		IF NOT WriteAdsPara.BUSY
			AND NOT WriteAdsPara.WRITE
		 	AND NOT Error
		THEN
			IF (forceSoftLimit XOR status.0) OR NOT InitDone.0 THEN
				InitDone.0 									:= TRUE;
				status.0 									:= forceSoftLimit;
				tmpWord 									:= BOOL_TO_UINT(forceSoftLimit);
				State 										:= 1;
				Busy 										:= TRUE;

			ELSIF(forceCalibration XOR status.1) OR NOT InitDone.1 THEN
				InitDone.1 									:= TRUE;
				status.1 									:= forceCalibration;
				tmpWord 									:= BOOL_TO_UINT(forceCalibration);
				State 										:= 10;
				Busy 										:= TRUE;
	
			ELSIF(forcePosLagMon XOR status.2) OR NOT InitDone.2 THEN
				InitDone.2 									:= TRUE;
				status.2 									:= forcePosLagMon;
				tmpWord 									:= BOOL_TO_UINT(forcePosLagMon);
				State 										:= 20;
				Busy 										:= TRUE;
			ELSIF(forcePosMon XOR status.3) OR NOT InitDone.3 THEN
				InitDone.3 									:= TRUE;
				status.3 									:= forcePosMon;
				tmpWord 									:= BOOL_TO_UINT(forcePosMon);
				State 										:= 30;
				Busy 										:= TRUE;
			ELSIF(forceTargetMon XOR status.4) OR NOT InitDone.4 THEN
				InitDone.4 									:= TRUE;
				status.4 									:= forceTargetMon;
				tmpWord 									:= BOOL_TO_UINT(forceTargetMon);
				State 										:= 40;
				Busy 										:= TRUE;
		
			END_IF
		ELSE
			WriteAdsPara	(Write := FALSE);
		END_IF

	1: (* toggle positive limit switches ****************************************************************)
		IF NOT WriteAdsPara.Busy
			AND WriteAdsPara.Write
		THEN
			IF WriteAdsPara.Err THEN
				State 										:= 9999;  // goto Error-state 
			ELSE           									
				State 										:= State + 1;
			END_IF         	
		END_IF

		WriteAdsPara(
			IdxGrp	:=16#4000+AxisId,
			IdxOffs	:=16#1000C,
			LEN		:=SIZEOF(tmpWord),
			SrcAddr	:=ADR(tmpWord),
			Write 	:= State = 1);

	2: (* toggle negative limit switches *****************************************************************)
		IF NOT WriteAdsPara.Busy
			AND WriteAdsPara.Write
		THEN
			IF WriteAdsPara.Err THEN
				State 										:= 9999; // goto Error-state 
			ELSE
				State 										:= 99; // done 
			END_IF
		END_IF

		WriteAdsPara(
			IdxGrp	:=16#4000+AxisId,
			IdxOffs	:=16#1000B,
			LEN		:=SIZEOF(tmpWord),
			SrcAddr	:=ADR(tmpWord),
			Write 	:= State = 2);

	10: (* set referenceflag *****************************************************************)
		IF NOT WriteAdsPara.Busy
			AND WriteAdsPara.Write
		THEN
			IF WriteAdsPara.Err THEN
				State 										:= 9999;  	// goto Error-state 
			ELSE           									
				State 										:= 99; 		// done 
			END_IF
		END_IF

		WriteAdsPara(
			IdxGrp	:=16#5100+AxisId,
			IdxOffs	:=16#9,
			LEN		:=SIZEOF(tmpWord),
			SrcAddr	:=ADR(tmpWord),
			Write 	:= State = 10 );
			
	20: (* lagdistance monitoring *****************************************************************)
		IF NOT WriteAdsPara.Busy
			AND WriteAdsPara.Write
		THEN
			IF WriteAdsPara.Err THEN
				State 										:= 9999;  	// goto Error-state 
			ELSE           									
				State 										:= 99; 		// done
			END_IF
		END_IF

		WriteAdsPara(
			IdxGrp	:=16#6000+AxisId,
			IdxOffs	:=16#10,
			LEN		:=SIZEOF(tmpWord),
			SrcAddr	:=ADR(tmpWord),
			Write 	:= State = 20);
			
	30: (* Position Monitoring *****************************************************************)
		IF NOT WriteAdsPara.Busy
			AND WriteAdsPara.Write
		THEN
			IF WriteAdsPara.Err THEN
				State 										:= 9999;  	// goto Error-state 
			ELSE           									
				State 										:= 99; 		// done
			END_IF
		END_IF

		WriteAdsPara(

			IdxGrp	:=16#4000+AxisId,
			IdxOffs	:=16#F,
			LEN		:=SIZEOF(tmpWord),
			SrcAddr	:=ADR(tmpWord),
			Write 	:= State = 30 );

	40: (* Target Monitoring *****************************************************************)
		IF NOT WriteAdsPara.Busy
			AND WriteAdsPara.Write
		THEN
			IF WriteAdsPara.Err THEN
				State 										:= 9999;  	// goto Error-state 
			ELSE           									
				State 										:= 99; 		// done
			END_IF
		END_IF

		WriteAdsPara(
			IdxGrp	:=16#4000+AxisId,
			IdxOffs	:=16#15,
			LEN		:=SIZEOF(tmpWord),
			SrcAddr	:=ADR(tmpWord),
			Write 	:= State = 40 );
			
	ELSE (* case else *)
		IF WriteAdsPara.ERR THEN
			Error											:= TRUE;
			ErrorID											:= WriteAdsPara.ERRID;
			LastErrText										:= CONCAT('Err WriteAdsPara ID: ', UDINT_TO_STRING(ErrorID));
		ELSE            									
			State 											:= 0;
		END_IF
	END_CASE
END_IF

(************************************************************************************************************************)

END_FUNCTION_BLOCK

// POUs/Motion/TF50xx-NC/03_Utilities/AxAutoWriteSoftLimit
{attribute 'no_check'}
FUNCTION_BLOCK AxAutoWriteSoftLimit
VAR_INPUT
	Enable													:	BOOL := FALSE; (* Enable Block *)
	AxId													: 	DWORD; (* ID der Achse *)
	SoftLimitPos											:	LREAL;
	SoftLimitNeg											:	LREAL;
END_VAR                         							
VAR_IN_OUT                      							
END_VAR                         							
VAR_OUTPUT        
	Busy													:	BOOL := FALSE;
	Error													:	BOOL := FALSE;
	{attribute 'displaymode':='hex'}  
	ErrorID													:	UDINT := 0;
END_VAR                         	
VAR
(* Cache **********************************************************************)
	State													: 	INT;
	MemLimitPos												:	LREAL;
	MemLimitNeg												:	LREAL;
	WriteReg												:	BYTE;

(* Instances *******************************************************************)
	WriteAdsPara											: 	ADSWRITE := (NetId	:= '' , Port := 500, TmOut	:= DEFAULT_ADS_TIMEOUT);

(* Dummy  *********************************************************************)
END_VAR

	(* Easy soft limit change 																		*)
	(************************************************************************************************)

(* writing parameters *******************************************************************************)
IF NOT Enable 
THEN
	MemLimitPos												:= SoftLimitPos;
	MemLimitNeg												:= SoftLimitNeg;
	                										
	State 													:= 0;
	Error													:= FALSE;
	ErrorID													:= 0;
	Busy 													:= FALSE;
ELSIF Axid = 0 
THEN
	ErrorID													:= E_AdsErr.DEVICE_INVALIDPARM;
	Error													:= FALSE;
	Busy													:= FALSE;
ELSE
	CASE State OF
	0:	(* Init *)

		Busy 												:= FALSE;

		IF NOT WriteAdsPara.BUSY
			AND NOT WriteAdsPara.WRITE
		 	AND NOT Error
		THEN
			WriteReg.0										:= SoftLimitPos <> MemLimitPos;
			WriteReg.1										:= SoftLimitNeg <> MemLimitNeg;
			
			IF WriteReg <> 0
			THEN
				Busy 										:= TRUE;
				state										:= state + SEL(WriteReg.0, 2, 1); //Jump to 2 if only negative changed
				MemLimitPos									:= SoftLimitPos;
				MemLimitNeg									:= SoftLimitNeg;
			END_IF
		ELSE
			WriteAdsPara	(Write := FALSE);
		END_IF

	1: (* Write positive limit to NC ****************************************************************)
		WriteAdsPara( Write := WriteReg.0, IdxGrp	:=16#4000+AxID, IdxOffs	:=16#1000E, LEN	:=SIZEOF(MemLimitPos), SrcAddr	:=ADR(MemLimitPos));	
		IF NOT WriteAdsPara.Busy
		THEN
			IF WriteAdsPara.Err 
			THEN
				ErrorId										:= WriteAdsPara.ERRID;
				Error										:= TRUE;
				Busy										:= FALSE;
				state										:= 0;
			ELSE           									
				State 										:= State + 1;
			END_IF   
			WriteAdsPara(Write := FALSE);      	
		END_IF


	2: (* Write negative limit to NC ****************************************************************)
		WriteAdsPara( Write := WriteReg.1, IdxGrp	:=16#4000+AxID, IdxOffs	:=16#1000D, LEN	:=SIZEOF(MemLimitNeg), SrcAddr	:=ADR(MemLimitNeg));	
		IF NOT WriteAdsPara.Busy
		THEN
			IF WriteAdsPara.Err 
			THEN
				ErrorId										:= WriteAdsPara.ERRID;
				Error										:= TRUE;
				Busy										:= FALSE;
				state										:= 0;
			ELSE           									
				State 										:= 0;
			END_IF   
			WriteAdsPara(Write := FALSE);      	
		END_IF
	END_CASE
END_IF

(************************************************************************************************************************)

END_FUNCTION_BLOCK

// POUs/Motion/TF50xx-NC/03_Utilities/AxCalcPosBias
{attribute 'no_check'}
//Calculates (new) NC axis position bias  
FUNCTION_BLOCK AxCalcPosBias EXTENDS FbBase
VAR_OUTPUT CONSTANT
//option settings 
	{attribute 'displaymode':='binary'}
	OPTION_WRITE_TO_NC										: 	BYTE :=2#0000_0001; //New position offset (bias) will directly written into the NC
END_VAR
VAR_INPUT
	{attribute 'displaymode':='binary'}
	Options													:	BYTE := 2#0000_0000; (* option constants are predefined, so they can accordingly be passed symbolically to the block *)
	SetPos													: 	LREAL := 0.0; //New actual positon of axis 
END_VAR
VAR_IN_OUT
	Axis													:	AXIS_REF;
END_VAR
VAR_OUTPUT
	RawPos													: LREAL; // Uncorrected axis position (Offset = 0.0)	
	Offset													: LREAL; // New postition offset (Position bias) 

END_VAR
VAR
(*  Memory *****************************************************)
	LastErrorId												:	UDINT;
	LastErrorState											:	INT;

(*  Timer ******************************************************)


(*  Trigger ****************************************************)

(*  Blocks *****************************************************)
	ReadAdsPara												: ADSREAD := (NetID:= '' , Port:=AMSPORT_R0_NC,TmOut := DEFAULT_ADS_TIMEOUT );
	WriteAdsPara											: ADSWRITE := (NetID:= '' , Port:=AMSPORT_R0_NC,TmOut := DEFAULT_ADS_TIMEOUT );

(*  Error ******************************************************)
(*  Dummys *****************************************************)
	{attribute 'hide' := ''}
END_VAR

	(* Calculate new pos bias (position offset)			 	 *)
	(*********************************************************)
	
(* Sequence ********************************************************)

	rtExecute(CLK := Execute);
	CASE state OF
	0 : 
		Busy 												:= FALSE;
		IF NOT Execute THEN
			Done 											:= FALSE;
			Error 											:= FALSE;
			ErrorID 										:= 0;
		END_IF
		IF rtExecute.Q THEN
			ReadAdsPara( Read := FALSE ); 
			WriteAdsPara(Write := FALSE);
			Busy											:= TRUE;
			Offset											:= 0.0;
			RawPos											:= 0.0;
			Done 											:= FALSE;
			Error 											:= FALSE;
			ErrorID 										:= 0;
			state 											:= state + 1;
		END_IF
		
		
	(* Read current pos. bias **********************************************)
	1:
		ReadAdsPara(Read:= TRUE,	IDxGrp:=(16#5000+Axis.NcToPlc.AxisId) , IDxOffs:=16#7,LEN:=SIZEOF(Offset), DestAddr:=ADR(Offset));	
		IF NOT ReadAdsPara.BUSY
		THEN
			IF ReadAdsPara.ERR
			THEN
				Busy										:= FALSE;
				Error										:= TRUE;
				ErrorID										:= ReadAdsPara.ERRID;
				LastErrorState								:= state;
				LastErrorId									:= ErrorId;
				state										:= 0;
			ELSE //Calculate new Pos bias
				RawPos										:= Axis.NcToPlc.ActPos - Offset;	
				Offset										:= SetPos - RawPos;
				IF (OPTION_WRITE_TO_NC AND Options) > 0
				THEN
					state									:= state + 1;
				ELSE
					Busy									:= FALSE;
					Done									:= TRUE;
					state									:= 0;					
				END_IF
			END_IF
		END_IF
		
	2:
		WriteAdsPara(Write:= TRUE,	IDxGrp:=(16#5000+Axis.NcToPlc.AxisId) , IDxOffs:=16#7,LEN:=SIZEOF(Offset), SrcAddr:=ADR(Offset));	
		IF NOT WriteAdsPara.BUSY
		THEN
			IF WriteAdsPara.ERR
			THEN
				Busy										:= FALSE;
				Error										:= TRUE;
				ErrorID										:= WriteAdsPara.ERRID;
				LastErrorId									:= ErrorId;
				LastErrorState								:= state;
				state										:= 0;
			ELSE			
				Busy										:= FALSE;
				Done										:= TRUE;
				state										:= 0;					
			END_IF
		END_IF		
	END_CASE

(****************************************************************************************)

PROPERTY PUBLIC optWritePosBiasToNC : BOOL
GET
optWritePosBiasToNC := Options.0;
END_GET
SET
Options.0 := optWritePosBiasToNC;
END_SET
END_PROPERTY

END_FUNCTION_BLOCK

// POUs/Motion/TF50xx-NC/03_Utilities/AxSoftSyncDistance
//Use this FB if NC-Reference mode is set to "Software Sync" or "Hardware-Sync".
//It is mandatory that the NC encoder parameter "Encoder Sub Mask (absolute range maximum value)" is set to the correct value!
//
//This FB checks the disctance between the falling edge of an reference sensor 
//and the final reference flag of the encoder (e.g. SingleTurn overflow in mode SoftwareSync)
//In case these two signals are very close together, it might be possible that the reference position varied about one motor turn
//depending whether the falling edge of the reference sensor occured before or after the software sync impulse.
//
//The FB reports an OK if the resulting distance if greater or equel than the "MinDistanceInDeg". 
{attribute 'no_check'}
FUNCTION_BLOCK AxSoftSyncDistance EXTENDS FbBase
VAR_OUTPUT CONSTANT
//option settings 
END_VAR
VAR CONSTANT
	DEG_PER_TURN											:	LREAL := 360.0;	
END_VAR
VAR_INPUT
	MinDistanceInDeg										:	LREAL := 45.0; //Minmum required distance between falling edge of sensor and software sync reference impuls (Single turn overflow)   
END_VAR
VAR_IN_OUT
	Axis													:	AXIS_REF;
END_VAR
VAR_OUTPUT
	Distance												: LREAL; //In user units (e.g. mm)
	DistancePerTurn											: LREAL; //In user units (e.g. mm)
	DistanceInDeg											: LREAL; //Resulting distance in degrees	
	OK														: BOOL;  //Inidcates whether the distance between falling edge of sensor and software sync is greater or equal than MinDistanceInDeg  
END_VAR
VAR
(*  Memory *****************************************************)
	LastErrorState											:	INT;
	LastErrorId												:	UDINT;
	ScalingNumerator										:	LREAL;
	ScalingDenumerator										:	LREAL;
	Scaling													:	LREAL;
	RefSystem												:	UDINT;
	RefMode													:	UDINT;
	{attribute 'displaymode':='hex'}
	EncSubMask												:	UDINT;


(*  Timer ******************************************************)

(*  Trigger ****************************************************)

(*  Blocks *****************************************************)
	ReadAdsPara												: ADSREAD := (NetID:= '' , Port:=AMSPORT_R0_NC,TmOut := DEFAULT_ADS_TIMEOUT );

(*  Error ******************************************************)
(*  Dummys *****************************************************)
	{attribute 'hide' := ''}
END_VAR

	(* Check distance between falling edge of reference sensor and deteced sync impulse		*)
	(****************************************************************************************)
	
(* Sequence ********************************************************)
	rtExecute(CLK := Execute);
	CASE state OF
	0 : 
		Busy 												:= FALSE;
		IF NOT Execute THEN
			OK												:= FALSE;
			Done 											:= FALSE;
			Error 											:= FALSE;
			ErrorID 										:= 0;
		END_IF
		IF rtExecute.Q THEN
			ReadAdsPara( Read := FALSE); 
			Busy											:= TRUE;
			Distance										:= 0.0;
			ScalingNumerator								:= 0.0;
			ScalingDenumerator								:= 0.0;
			Scaling											:= 0.0;
			RefSystem										:= 0;
			EncSubMask										:= 0;
			OK												:= FALSE;
			Done 											:= FALSE;
			Error 											:= FALSE;
			ErrorID 										:= 0;
			state 											:= state + 1;
		END_IF
		
		
	(* Read scaling numerator **********************************************)
	1:
		ReadAdsPara(Read:= TRUE,	IDxGrp:=(16#5000+Axis.NcToPlc.AxisId) , IDxOffs:=16#23,LEN:=SIZEOF(ScalingNumerator), DestAddr:=ADR(ScalingNumerator));	
		IF NOT ReadAdsPara.BUSY
		THEN
			IF ReadAdsPara.ERR
			THEN
				Busy										:= FALSE;
				Error										:= TRUE;
				ErrorID										:= ReadAdsPara.ERRID;
				LastErrorState								:= state;
				LastErrorId									:= ErrorId;
				state										:= 0;
			ELSE 
				state										:= state + 1;						
			END_IF
			ReadAdsPara( Read := FALSE);
		END_IF
		
	(* Read scaling denumerator **********************************************)
	2:
		ReadAdsPara(Read:= TRUE,	IDxGrp:=(16#5000+Axis.NcToPlc.AxisId) , IDxOffs:=16#24,LEN:=SIZEOF(ScalingDenumerator), DestAddr:=ADR(ScalingDenumerator));	
		IF NOT ReadAdsPara.BUSY
		THEN
			IF ReadAdsPara.ERR
			THEN
				Busy										:= FALSE;
				Error										:= TRUE;
				ErrorID										:= ReadAdsPara.ERRID;
				LastErrorState									:= state;
				LastErrorId									:= ErrorId;
				state										:= 0;
			ELSE
				Scaling										:= ScalingNumerator / SEL(ScalingDenumerator = 0.0, ScalingDenumerator , 1.0);	
				IF Scaling = 0.0
				THEN
					Busy									:= FALSE;
					Error									:= TRUE;
					ErrorID									:= MC_ERROR_PARAMETER_NOT_CORRECT;
					LastErrorState								:= state;
					LastErrorId									:= ErrorId;
					state									:= 0;	
				ELSE
					state									:= state + 1;
				END_IF					
			END_IF
			ReadAdsPara( Read := FALSE);
		END_IF

	(* Read distance in user units **********************************************)
	3:
		ReadAdsPara(Read:= TRUE,	IDxGrp:=(16#5100+Axis.NcToPlc.AxisId) , IDxOffs:=16#101,LEN:=SIZEOF(Distance), DestAddr:=ADR(Distance));	
		IF NOT ReadAdsPara.BUSY
		THEN
			IF ReadAdsPara.ERR
			THEN
				Busy										:= FALSE;
				Error										:= TRUE;
				ErrorID										:= ReadAdsPara.ERRID;
				LastErrorState									:= state;
				LastErrorId									:= ErrorId;
				state										:= 0;
			ELSE 
				state										:= state + 1;			
			END_IF
			ReadAdsPara( Read := FALSE);
		END_IF
		
	(* Read selected reference system **********************************************)
	4:
		ReadAdsPara(Read:= TRUE,	IDxGrp:=(16#5000+Axis.NcToPlc.AxisId) , IDxOffs:=16#19,LEN:=SIZEOF(RefSystem), DestAddr:=ADR(RefSystem));	
		IF NOT ReadAdsPara.BUSY
		THEN
			IF ReadAdsPara.ERR
			THEN
				Busy										:= FALSE;
				Error										:= TRUE;
				ErrorID										:= ReadAdsPara.ERRID;
				LastErrorState									:= state;
				LastErrorId									:= ErrorId;
				state										:= 0;
			ELSE 
				state										:= state + 1;					
			END_IF
			ReadAdsPara( Read := FALSE);
		END_IF
	
	(* Read selected reference mode **********************************************)
	5:
		ReadAdsPara(Read:= TRUE,	IDxGrp:=(16#5000+Axis.NcToPlc.AxisId) , IDxOffs:=16#107,LEN:=SIZEOF(RefMode), DestAddr:=ADR(RefMode));	
		IF NOT ReadAdsPara.BUSY
		THEN
			IF ReadAdsPara.ERR
			THEN
				Busy										:= FALSE;
				Error										:= TRUE;
				ErrorID										:= ReadAdsPara.ERRID;
				LastErrorState									:= state;
				LastErrorId									:= ErrorId;
				state										:= 0;
			ELSE 
				state										:= state + 1;					
			END_IF
			ReadAdsPara( Read := FALSE);
		END_IF
	
	(* Read EncSubMask (Inc per turn) **********************************************)
	6:
		ReadAdsPara(Read:= TRUE,	IDxGrp:=(16#5000+Axis.NcToPlc.AxisId) , IDxOffs:=16#108,LEN:=SIZEOF(EncSubMask), DestAddr:=ADR(EncSubMask));	
		IF NOT ReadAdsPara.BUSY
		THEN
			IF ReadAdsPara.ERR
			THEN
				Busy										:= FALSE;
				Error										:= TRUE;
				ErrorID										:= ReadAdsPara.ERRID;
				LastErrorState									:= state;
				LastErrorId									:= ErrorId;
				state										:= 0;
			ELSIF EncSubMask = 0
			THEN
				Busy										:= FALSE;
				Error										:= TRUE;
				ErrorID										:= MC_ERROR_PARAMETER_NOT_CORRECT;
				LastErrorState									:= state;
				LastErrorId									:= ErrorId;
				state										:= 0;			
			ELSE
				state										:= state + 1;					
			END_IF
			ReadAdsPara( Read := FALSE);
		END_IF
		
	(* Check reference value ************************************)
	7:
		DistancePerTurn										:= EncSubMask * Scaling;
		DistanceInDeg										:= (DEG_PER_TURN / DistancePerTurn) * Distance;	
																		
		OK													:= ABS(DistanceInDeg) <= DEG_PER_TURN - ABS(MinDistanceInDeg)  
																AND ABS(DistanceInDeg) >= ABS(MinDistanceInDeg) ;							
	
		Busy												:= FALSE;
		Done												:= TRUE;
		state												:= 0;	
	END_CASE

(****************************************************************************************)

END_FUNCTION_BLOCK

// POUs/Motion/TF50xx-NC/03_Utilities/AxStatemodel
{attribute 'no_check'}
//based on Statemodel instance
//IMPORTANT call this functionblock after AxAdmin !!!!
FUNCTION_BLOCK AxStatemodel EXTENDS Statemodel_Unit
VAR_INPUT 
	PT_DelEStopDisableAx									:	TIME := T#800MS;
	SafetyOK												:	BOOL := TRUE; //Drive safety card OK
	ENSoEReset												:	BOOL := TRUE;
	ErrorActive												:	BOOL := FALSE; //Axis in error	
	Dec														:	LREAL := 0.0;
	Jerk													:	LREAL := 0.0;
	rAxis													:	REFERENCE TO AXIS_REF := 0;
END_VAR
VAR_OUTPUT
END_VAR
VAR
	MC_Stop													: 	MC_Stop;
	MC_Reset												:	MC_Reset;
	SOE_Reset												:	FB_SoEReset;
	Mainstate												:	INT := 0;
	Ton_Seq													:	TON;
{attribute 'displaymode':='binary'}
	MemAbortingStep											:	BYTE; //Show online reasons for the aporting steps
END_VAR

	(* Axis UnitStateCtrl				 		V1.3		*)
	(*														*)
	(********************************************************)

(* check rAxis ************************************************)
IF NOT __ISVALIDREF(rAxis) 
THEN 
(*	ErrorText			:= 'Pointer pAxis invalid (0)'; *)
	RETURN;
END_IF

(* work local sub ****************************************)
	unit.name			:= CONCAT('Unit Axis ID: ', UDINT_TO_STRING(rAxis.NcToPlc.AxisId));

(* Call super ***************************************)
	SUPER^(); //Execute generic unit
		
(*********************************************************)

METHOD PROTECTED aborted : BOOL //Return value = TRUE if execution finsihed
VAR_INPUT
END_VAR
rAxis.PlcToNc.ControlDWord.0 						:= FALSE; (* Enable *)
rAxis.PlcToNc.ControlDWord.1 						:= FALSE; (* Enable_Positive *)
rAxis.PlcToNc.ControlDWord.2 						:= FALSE; (* Enable_Negative *)

MC_Stop(
	Axis			:= rAxis,
	Execute			:= 	MC_Stop.Execute 
						AND F_AxisControlLoopClosed(stateDWord := rAxis.NcToPlc.stateDWord) 
						AND rAxis.Status.PTPmode ,  (* Block new motion cmd *)
	Deceleration	:= ,
	Jerk			:= ,
	Options			:= ,
	Done			=> ,
	Busy			=> ,
	Active			=> ,
	CommandAborted	=> ,
	Error			=> ,
	ErrorID			=> );
	
Aborted												:= NOT MC_Stop.Done or MC_Stop.Error;
END_METHOD

METHOD PROTECTED aborting : BOOL //Return value = TRUE if execution finsihed
VAR_INPUT
END_VAR
CASE Mainstate OF
		0: (* Step 1 -> start stopping *)
			Ton_Seq(IN := FALSE , PT := PT_DelEStopDisableAx);
			MemAbortingStep									:= 0;
			IF NOT rAxis.Status.PTPmode
				OR rAxis.Status.ProtectedMode
				OR rAxis.Status.MotionCommandsLocked
				OR NOT rAxis.Status.Operational
			THEN (* axis is slave-axis *)
				Mainstate									:= 99;
				MemAbortingStep.7							:= TRUE; 
			ELSIF NOT MC_Stop.busy      					
			THEN                        					
				MemAbortingStep.1							:= TRUE;
				Mainstate									:= 1;
			END_IF


			MC_Stop(
				Axis			:= rAxis,
				Execute			:= Mainstate = 1 AND NOT rAxis.Status.Decelerating ,
				Deceleration	:=  Dec,(* NOT-HALT Parameter uebergeben *)
				Jerk			:= Jerk, (* NOT-HALT Parameter uebergeben *)
				Options			:= ,
				Done			=> ,
				Busy			=> ,
				Active			=> ,
				CommandAborted	=> ,
				Error			=> ,
				ErrorID			=> );

		1: (* Step 2 -> if stopped or safety signal = FALSE *) 
			MC_Stop(
				Axis			:= rAxis,
				Execute			:= ,
				Deceleration	:= ,
				Jerk			:= ,
				Options			:= ,
				Done			=> ,
				Busy			=> ,
				Active			=> ,
				CommandAborted	=> ,
				Error			=> ,
				ErrorID			=> );

			Ton_Seq(IN := TRUE);
			IF rAxis.Status.Decelerating 
			THEN
				MemAbortingStep.2							:= TRUE;
				Mainstate									:= 99;
			ELSIF rAxis.Status.NotMoving					
			THEN                        					
				MemAbortingStep.3							:= TRUE;
				Mainstate									:= 99;
			ELSIF Ton_Seq.Q             					
			THEN                        					
				MemAbortingStep.6							:= TRUE;
				Mainstate									:= 99;
			END_IF
	
		99: (* disable feed *)		
			rAxis.PlcToNc.ControlDWord.1 					:= FALSE; (* Enable_Positive *)
			rAxis.PlcToNc.ControlDWord.2 					:= FALSE; (* Enable_Negative *)
			Ton_Seq(IN := TRUE);         					
			IF rAxis.Status.NotMoving 
				OR Ton_Seq.Q
			THEN
				MemAbortingStep.4							:=  rAxis.Status.NotMoving;
				Unit.StateComplete();
			END_IF
			Aborting										:= TRUE;
		END_CASE
END_METHOD

METHOD PROTECTED clearing : BOOL //Return value = TRUE if execution finsihed
VAR_INPUT
END_VAR
CASE Mainstate OF
0:
	MC_Stop(
		Axis			:= rAxis,
		Execute			:= FALSE,
		Deceleration	:= , 
		Jerk			:= , 
		Options			:= , 
		Done			=> , 
		Busy			=> , 
		Active			=> , 
		CommandAborted	=> , 
		Error			=> , 
		ErrorID			=> );
		
	IF NOT MC_Stop.Busy
	THEN
		Mainstate									:= 99;
	END_IF
				
99:
	IF NOT rAxis.PlcToNc.ControlDWord.0 (* Enable is already active *)
		OR F_AxisControlLoopClosed(stateDWord := rAxis.NcToPlc.stateDWord)
		OR ErrorActive
	THEN
		Clearing									:= TRUE;
		Unit.StateComplete();
	END_IF
			
END_CASE
END_METHOD

METHOD PROTECTED completing : Bool //Return value = TRUE if execution finsihed
VAR_INPUT
END_VAR
(* Fehler ausloesen *)
IF UNit.InCompleting
	AND NOT F_AxisHasJob(stateDWord := rAxis.NcToPlc.stateDWord)
THEN
	Unit.StateComplete();
	Completing											:= TRUE;
ELSE
	Completing 											:= Executing();
END_IF
END_METHOD

METHOD PROTECTED executing : booL
VAR_INPUT
END_VAR
(* Set statemodel to error if axis is in error *********)
IF rAxis.NcToPlc.ErrorCode <> 0 OR ErrorActive 
THEN
	IF unit.optEnableFwdMachineErrorToMaster
	THEN
		Unit.SetMachineError();
	ELSE
		Unit.SetLocalError();
	END_IF
END_IF
	
Executing 												:= Unit.isStateActive(Unit.State);
END_METHOD

METHOD PROTECTED resetting : Bool //Return value = TRUE if execution finsihed
VAR_INPUT
END_VAR
		CASE Mainstate OF
		0:
			Ton_Seq(IN := FALSE);
			
			MC_Reset(
				Axis		:= rAxis,
				Execute		:= FALSE);
				
			SOE_Reset(
				Axis		:= rAxis,
				Execute		:= FALSE);

			IF SOE_Reset.Busy
				OR MC_Reset.Busy
			THEN
				;
			ELSIF SafetyOK
			THEN
				Mainstate									:= 10;
			ELSE            								
				Mainstate									:= 1;
			END_IF          	

		1: (* Wartezeit bis Safety OK *)
			Ton_Seq(IN := TRUE, PT := T#3S);
			IF SafetyOK	
			THEN
				Mainstate									:= 2;
			ELSIF Ton_Seq.Q 
			THEN (* Karten nicht resetbar .... *)
				Ton_Seq(IN := FALSE);
				Mainstate									:= 10;
			END_IF
			

		2: (* Wartezeit nach Safety Reset *)
			Ton_Seq(IN :=TRUE, PT := T#100MS);
			IF Ton_Seq.Q
			THEN
				Ton_Seq(IN := FALSE);
				Mainstate									:= 10;
			END_IF

		10: 
			SOE_Reset(
				Axis	:= rAxis,
				Execute	:= ENSoEReset AND(rAxis.Status.Error OR rAxis.Status.DriveDeviceError));

			Mainstate										:= 11;

		11:
			SOE_Reset(Axis	:= rAxis);
			IF NOT SOE_Reset.Busy THEN
				Mainstate			:= 20;
			END_IF

		20:
			MC_Reset(
				Axis	:= rAxis,
				Execute	:= NOT rAxis.Status.ProtectedMode OR rAxis.Status.Error);

			Mainstate										:= 21;

		21:
			MC_Reset( Axis	:= rAxis);
			IF NOT MC_Reset.Busy 
			THEN
				Mainstate									:= 99;
				Ton_Seq(IN := FALSE);
			END_IF

		99:
			Ton_Seq(IN := TRUE, PT := T#3S);
			MC_Reset(
				Axis	:= rAxis,
				Execute	:= FALSE);
				
			SOE_Reset(
				Axis	:= rAxis,
				Execute	:= FALSE);

			IF NOT MC_Reset.Busy
				AND NOT SOE_Reset.Busy
				AND(Ton_Seq.Q OR NOT ErrorActive AND NOT rAxis.Status.Error) 
			THEN
				Unit.StateComplete();
				Resetting									:= TRUE;
			END_IF
		END_CASE
END_METHOD

METHOD PROTECTED starting : Bool
VAR_INPUT
END_VAR
Unit.StateComplete();
Starting													:= Executing();
END_METHOD

METHOD PROTECTED stopped : Bool //Return value = TRUE if execution finsihed
VAR_INPUT
END_VAR
		MC_Stop(
			Axis			:= rAxis,
			Execute			:= FALSE,
			Deceleration	:= ,
			Jerk			:= ,
			Options			:= ,
			Done			=> ,
			Busy			=> ,
			Active			=> ,
			CommandAborted	=> ,
			Error			=> ,
			ErrorID			=> );
			
		Stopped													:= MC_Stop.Done OR MC_Stop.Error;
END_METHOD

METHOD PROTECTED stopping : BOOL //Return value = TRUE if execution finsihed
VAR_INPUT
END_VAR
		CASE Mainstate OF
		0:
			IF NOT MC_Stop.busy
			THEN
				Mainstate									:= 1;
			END_IF		

			MC_Stop(
				Axis			:= rAxis,
				Execute			:= 	Mainstate <> 0 
									AND NOT rAxis.Status.ProtectedMode 
									AND rAxis.Status.PTPmode,
				Deceleration	:= ,
				Jerk			:= ,
				Options			:= ,
				Done			=> ,
				Busy			=> ,
				Active			=> ,
				CommandAborted	=> ,
				Error			=> ,
				ErrorID		=> );

		1:
			MC_Stop(
				Axis			:= rAxis,
				Execute			:= 	MC_Stop.Execute 
									AND NOT rAxis.Status.NotMoving 
									AND rAxis.Status.ControlLoopClosed, (* Not Moving or not Operational *)
				Deceleration	:= ,
				Jerk			:= ,
				Options			:= ,
				Done			=> ,
				Busy			=> ,
				Active			=> ,
				CommandAborted	=> ,
				Error			=> ,
				ErrorID			=> );

			IF NOT MC_Stop.Execute 
			THEN
				Mainstate									:= 99;				
			END_IF
			
		99:
			Unit.StateComplete();
			Stopping										:= TRUE;
		END_CASE
END_METHOD

END_FUNCTION_BLOCK

// POUs/Statemodel/control/Statemodel
{attribute 'no_check'}
//Mode-Statemodel controller - inspired by OMAC statemodel
//FB is able to synchronize subordinate statemodel instances as well to be a subordinate instance at the same time 
//
//				(Line control SM)
//				I				I
//			(Feeder)			(Stacker)
//			I	 	I			I		I					
//		(XYAxis) (Belts)	(XYAxis) (Belts)		
//
{attribute 'reflection'} 
FUNCTION_BLOCK Statemodel IMPLEMENTS I_Statemodel
VAR_OUTPUT CONSTANT         								
	VERSION													:	STRING(5) := 'V6';
	MIN_SLAVE												:	INT := 1;	 
	MAX_SLAVE												:	INT := PARAM.STATEMODEL_CTRL_MAX_SLAVE; //see library parameter to customize parameter	
                     
//Statemodel error codes       								
	ERROR_MACHINE											:	INT := 1;	(* Error requested in reason of fatal machine error, all subs in then same unit change their state to Stopping with error *)
	ERROR_LOCAL												:	INT := 2; 	(* Error requested from this sub *)
	ERROR_EXTERNAL											:	INT := 3; 	(* Error requested by Unit in reason of fatal machine error in other Sub *)
{attribute 'displaymode':='binary'}
	OPTION_ENABLE_MODE_SWITCH_TO_IDLE						:	BYTE := 2#0000_0001; //Mode switched to Idle automatically if state Aborted/Stopped reached - as default the mode will not change
{attribute 'displaymode':='binary'}
	OPTION_ENABLE_MODE_CHANGE_IN_EXECUTE					:	BYTE := 2#0000_0010; //Mode change in state Execute, FALSE = mode change over state stopping
{attribute 'displaymode':='binary'}
	OPTION_ENABLE_EXTERNAL_STATE_COMPLETE					:	BYTE := 2#0000_0100; //Default:Enable external use of method "StateComplete"! even if instance is controlling subs as well
{attribute 'displaymode':='binary'}	
	OPTION_DISABLE_LOCAL_ESTOP								:	BYTE := 2#0000_1000; //Disable local EStop signals, if sub ist remote controlled 
{attribute 'displaymode':='binary'}
	OPTION_ENABLE_MASCHINE_ERROR_TO_MASTER					:	BYTE := 2#0001_0000; //Default:Machine error to remote master - With FALSE, a machine error  will not further up reported to the master
{attribute 'displaymode':='binary'}
	OPTION_ENABLE_MODE_CHANGE_VIA_STATE_COMPL				:	BYTE := 2#0010_0000; //Default:Mode change over state Completing - The statemodel switches to state "Completing" as an reaction of a new SetMode
{attribute 'displaymode':='binary'}
	OPTION_ENABLE_EXPLICIT_ERROR_RESET						:	BYTE := 2#0100_0000; //Default:Hold state Stopped until error is eplicit reseted with reset - instance stays at Stopped until error will be reset, even if the remote master change into reset 
{attribute 'hide'}
{attribute 'displaymode':='binary'}	
	OPTION_RESERVED											:	BYTE := 2#1000_0000; //not used
END_VAR
VAR_INPUT                   							
    {attribute 'instance-path'} 
    {attribute 'noinit'} 	
	Name													:	STRING;
{attribute 'displaymode':='binary'}
	Options													:	BYTE := 	2#0000_0000
																		//	OR OPTION_ENABLE_MODE_SWITCH_TO_IDLE		//Mode switched to Idle automatically if state Aborted/Stopped reached - as default the mode will not change
																		//	OR OPTION_ENABLE_MODE_CHANGE_IN_EXECUTE		//Mode change in state Execute, FALSE = mode change over state stopping
																			OR OPTION_ENABLE_EXTERNAL_STATE_COMPLETE	//Default:Enable external use of method "StateComplete"! even if instance is controlling subs as well
																		//	OR OPTION_DISABLE_LOCAL_ESTOP				//Disable local EStop signals, if sub ist remote controlled 
																			OR OPTION_ENABLE_MASCHINE_ERROR_TO_MASTER	//Default:Machine error to remote master - With FALSE, a machine error  will not further up reported to the master
																			OR OPTION_ENABLE_MODE_CHANGE_VIA_STATE_COMPL//Default:Mode change over state Completing - The statemodel switches to state "Completing" as an reaction of a new SetMode
																			OR OPTION_ENABLE_EXPLICIT_ERROR_RESET		//Default:Hold state Stopped until error is eplicit reseted with reset - instance stays at Stopped until error will be reset, even if the remote master change into reset 
																		//	OR OPTION_RESERVED							//not used
																			;		
(* Unit Safety Signals *)   								
	EStopDirectOK											:	BOOL := TRUE; (* -> Aborting *)
	EStopDelayOK											:	BOOL := TRUE; (* -> Aborted *)
	EStopOK													:	BOOL := TRUE; (* -> Clearing after EStop/Circuit OK *)
                            								
(* Signals *)               								
	ResetTrig												:	BOOL := FALSE; //Acknowledge/reset error - send also to subordinate instances  
	SetMode													:	eMODE := eMODE.IDLE; //Requested mode if instance is not a subordinate instance (RemotCtrlEnable = FALSE)
                            								
(* Remote UnitCtrl *)       								
	RemoteCtrlEnable										:	BOOL := TRUE;	//Statemodel follows remote master 
																						                           	
(* Sub Units - RemoteData from slave units *)
	ipSlave													:	ARRAY[MIN_SLAVE..MAX_SLAVE] OF I_Statemodel; (* RemoteData from slave units - WRITE THE ADRESS CYCLIC!! *)
END_VAR
VAR_OUTPUT
	Id														:	INT; //Unique Id for each statemodel instance
	IdRemoteMaster											:	INT; //Id of remote master 
	Info													:	STRING(30) := 'eSTATE.STARTUP'; //State name as string
	Busy													:	BOOL := TRUE; //Will be set to true as a result of a state change - set to false with method "StateComplete" to 
	SlavesInSync											:	BOOL; //local statemodel and subordinate (external) subs state are equel 
	SlavesBusy												:	BOOL; //minimum one sub is still busy - not complete
	NoOfBusySlaves											:	INT;	
	Mode													:	eMODE := eMODE.IDLE ;  //Active mode 
	State													:	eSTATE := eSTATE.STARTUP;//Active state
	EStopStartupOK											:	BOOL;	//EStop/Circuit is ok (clearing done)
	RT_StateChanged 										:	BOOL; //Rising flag to signal a state change
	(* StateBits *)         								
	InStartup												:	BOOL := TRUE; 	
	InIdle													:	BOOL ;
	InStarting												:	BOOL ;
	InStarted												:	BOOL ;
	InExecute												:	BOOL ;
	InCompleting											:	BOOL ;
	InComplete												:	BOOL ;
	InAborting												:	BOOL ;
	InAborted												:	BOOL ;
	InClearing												:	BOOL ;
	InStopping												:	BOOL ;
	InStopped												:	BOOL ;
	InResetting												:	BOOL ;
                            								   
(* optional not in use  										
	InHolding												:	BOOL := False;
	InHeld													:	BOOL := False;
	InUnholding												:	BOOL := False;
	InSuspending											:	BOOL := False;
	InSuspended												:	BOOL := False;
	InUnsuspending											:	BOOL := False;
*)       
	ErrHdl													:	ERROR_HDL;
                   								
END_VAR                     								
VAR
(* cache ********************************************)
	LastState												:	eSTATE := eSTATE.STARTUP;
	GoToAborting											:	BOOL ;
	Localreset												:	BOOL ;
	Remotereset												:	BOOL ;
	BusyIntern												:	BOOL := TRUE;
                          								
	(* Remote Data *)       								
	MasterCmdMode											:	eMODE; //Mode commanded from Master through remote data property
	MasterCmdState											:	eSTATE; //State commanded from Master through remote data property
	MasterCmdInfo											:	WORD; (* Info data from master through remote data property
																		Bit 0-7 = Options																	
																		Bit 8 = RemoteCtrlEnable
																		Bit 9 = Ack 
																		Bit 10 = Busy
																		Bit 11 = ErrorMaschine
																		Bit 12 = ErrorLocal 
																		Bit 13 = ErrorExternal 
																		Bit 14 = EStopOK
																		Bit 15 = EStopDelayOK *) 
   	RemoteDataToSlaves										:	U_64BIT_DATATYPE;
   	RemoteDataFromSlave										:	U_64BIT_DATATYPE;
																			
 	(* Sync Sub Status *)   								
	NoSlavesConnected										:	BOOL ; (* no external subs (Pointer) in use *)
	SlavesState												:	eSTATE := eSTATE.STARTUP; (* summary states from SubCtrls *)
 
(* function-blocks ******************************************************)
	GetTaskIndex 											: 	GETCURTASKINDEX;

(* internal used variables **********************************************)                       								
	i														: INT := 0 ;
END_VAR

(* Unit mode model - statemachine			- view constant -	*)
(****************************************************************)

(*******************************************************'********)
(* Init Pointer in First Cycle 									*)
(****************************************************************)

(* Init state model instance **************************************)
	IF GetTaskIndex.index = 0 THEN GetTaskIndex();  END_IF
	IF TwinCAT_SystemInfoVarList._TaskInfo[GetTaskIndex.Index].FirstCycle 
	THEN
		RETURN;		
	END_IF
		
(* Set Local ack *********************************************)
	RemoteReset 											:= MasterCmdInfo.9;
	LocalReset 												:= ResetTrig OR RemoteReset OR LocalReset;

(* work Busy if no external subs in use ****************************************)
	IF NoSlavesConnected AND NOT Options.2 
	THEN 
		BusyIntern 											:= FALSE; 
	END_IF (* no subs and no external StateCompl *)
	
	IF NoSlavesConnected AND NOT BusyIntern 
	THEN 
		Busy 												:= NOT EStopOK AND NOT Options.3 AND InClearing; 
	END_IF

(* Signals ************************************************)
	GoToAborting											:=(	NOT RemoteCtrlEnable OR NOT Options.3)
																AND (NOT EStopDirectOK OR NOT EStopDelayOK)
																OR
																RemoteCtrlEnable
																AND (MasterCmdState = eSTATE.ABORTING OR MasterCmdState = eSTATE.ABORTED);

(* Local State Machine ****************************************************)
	CASE State OF
	{region "STARTUP"} 
	eSTATE.STARTUP: info 									:= TO_STRING(eSTATE.STARTUP);
	
		IF NOT Busy 
		THEN (* Busy initalisation is TRUE *)
			Busy := BusyIntern 								:= TRUE;
			state 											:= eSTATE.ABORTING;
		ELSE
			; (* Wait for Startup End*)
		END_IF
	{endregion} 		
	{region "IDLE"} 
	eSTATE.IDLE:
		info 												:= TO_STRING(eSTATE.IDLE);
		
		IF GoToAborting 
		THEN
			Busy := BusyIntern 								:= TRUE; 
			state 											:= eSTATE.ABORTING;
		ELSIF RemoteCtrlEnable AND MasterCmdState = eSTATE.STOPPING 
		THEN
			Busy := BusyIntern 								:= TRUE; 
			state 											:= eSTATE.STOPPING;
		ELSIF NOT RemoteCtrlEnable AND SetMode <> eMODE.IDLE
			OR 
			RemoteCtrlEnable
			AND MasterCmdState <> eSTATE.IDLE
			AND MasterCmdState <> eSTATE.RESETTING
		THEN
			Busy := BusyIntern 								:= TRUE; 
			Mode 											:= SEL(RemoteCtrlEnable,SetMode,MasterCmdMode);
			State 											:= eSTATE.STARTING;
		ELSE
			Mode 											:= eMODE.IDLE;
		END_IF
	{endregion} 
	{region "STARTING"} 	
	eSTATE.STARTING: info 									:= TO_STRING(eSTATE.STARTING);
	
		IF GoToAborting 
		THEN
			state 											:= eSTATE.ABORTING;
			Busy := BusyIntern 								:= TRUE;

		ELSIF RemoteCtrlEnable
			AND(
			MasterCmdState = eSTATE.STOPPING
			OR (* Betriebsartenwechsel ueber RemoteCtrl ein *)
			NOT RemoteDataToSlaves._WORDS[2].8 AND Mode <> MasterCmdMode)
		THEN
			state 											:= eSTATE.STOPPING;
			Busy := BusyIntern 								:= TRUE;
		ELSIF NOT Busy 
		THEN
			state 											:= eSTATE.STARTED;			
		END_IF
	{endregion} 		
	{region "STARTED"} 	
	eSTATE.STARTED: info 									:= TO_STRING(eSTATE.STARTED);
		
		IF GoToAborting 
		THEN
			Busy := BusyIntern 								:= TRUE; 
			state 											:= eSTATE.ABORTING;
		ELSIF RemoteCtrlEnable
			AND NOT RemoteDataToSlaves._WORDS[2].8 
			AND Mode <> MasterCmdMode
		THEN (* Betriebsartenwechsel ueber RemoteCtrl ein *)
			Busy := BusyIntern 								:= TRUE; 
			state 											:= eSTATE.STOPPING;
		ELSIF NOT RemoteCtrlEnable
			OR 	
			RemoteCtrlEnable
			AND MasterCmdState <> eSTATE.STARTED
			AND MasterCmdState <> eSTATE.STARTING
		THEN
			IF RemoteCtrlEnable AND MasterCmdState = eSTATE.EXECUTE
				OR NOT RemoteCtrlEnable
			THEN
				Busy := BusyIntern 							:= TRUE; 
				state 										:= eSTATE.EXECUTE;
			ELSIF RemoteCtrlEnable AND Options.5 //Compl. aktiviert
				AND(MasterCmdState = eSTATE.COMPLETING OR	MasterCmdState = eSTATE.COMPLETE)
			THEN
				Busy := BusyIntern 							:= TRUE; 
				state 										:= eSTATE.COMPLETING;
			ELSE
				Busy := BusyIntern 							:= TRUE; 
				state 										:= eSTATE.STOPPING;
			END_IF
		END_IF
	{endregion} 	
	{region "EXECUTE"} 
	eSTATE.EXECUTE: info 									:= TO_STRING(eSTATE.EXECUTE);
	
		IF GoToAborting 
		THEN
			Busy := BusyIntern 								:= TRUE; 
			state 											:= eSTATE.ABORTING;

		ELSIF SetMode <> Mode
			AND NOT RemoteCtrlEnable
			AND NOT Options.1  (* Modewechsel ueber Stopping/Completing wenn Options.1 nicht gesetzt *)
			OR	
			NOT RemoteCtrlEnable
			AND SetMode = eMODE.IDLE
			OR	
			RemoteCtrlEnable
			AND MasterCmdState <> eSTATE.EXECUTE
			AND MasterCmdState <> eSTATE.STARTING
			AND MasterCmdState <> eSTATE.STARTED
			OR (* Betriebsartenwechsel ueber RemoteCtrl ein *)
			RemoteCtrlEnable
			AND NOT RemoteDataToSlaves._WORDS[2].8 AND Mode <> MasterCmdMode
		THEN
			IF Options.5 (* Mode change over Completing *)
				AND(MasterCmdState = eSTATE.COMPLETING
				AND RemoteCtrlEnable
				OR	
				NOT RemoteCtrlEnable)
			THEN
				Busy := BusyIntern 							:= TRUE; 
				state 										:= eSTATE.COMPLETING;
			ELSE      						
				Busy := BusyIntern 							:= TRUE; 				
				state 										:= eSTATE.STOPPING;
			END_IF

		ELSIF Options.1  (* Modewechsel in Execute *)
			AND(
			SetMode <> Mode AND NOT RemoteCtrlEnable
			OR	
			MasterCmdMode <> Mode AND RemoteCtrlEnable)
		THEN
			Mode 											:= SEL(RemoteCtrlEnable,SetMode,MasterCmdMode);

		ELSIF RemoteCtrlEnable
			AND(
			MasterCmdState = eSTATE.HOLDING 
			OR MasterCmdState = eSTATE.HELD) 
		THEN
			Busy := BusyIntern 								:= TRUE; 
			state 											:= eSTATE.HOLDING;
		ELSIF RemoteCtrlEnable
			AND(
			MasterCmdState = eSTATE.SUSPENDING 
			OR MasterCmdState = eSTATE.SUSPENDED) 
		THEN
			Busy := BusyIntern 								:= TRUE; 
			state 											:= eSTATE.SUSPENDING;
		END_IF
	{endregion} 	
	{region "SUSPENDING"} 
	eSTATE.SUSPENDING: 	info 								:= TO_STRING(eSTATE.SUSPENDING);	
		
		IF GoToAborting 
		THEN
			state 											:= eSTATE.ABORTING;
			Busy := BusyIntern 								:= TRUE;

		ELSIF RemoteCtrlEnable
			AND(
			MasterCmdState = eSTATE.STOPPING
			OR (* Betriebsartenwechsel ueber RemoteCtrl ein *)
			NOT RemoteDataToSlaves._WORDS[2].8 AND Mode <> MasterCmdMode)
		THEN
			state 											:= eSTATE.STOPPING;
			Busy := BusyIntern 								:= TRUE;
		ELSIF NOT Busy 
		THEN
			state 											:= eSTATE.SUSPENDED;		
		END_IF	
	{endregion} 	
	{region "SUSPENDED"} 
	eSTATE.SUSPENDED:	info 								:= TO_STRING(eSTATE.SUSPENDED);	
	
		IF GoToAborting 
		THEN
			Busy := BusyIntern 								:= TRUE; 
			state 											:= eSTATE.ABORTING;
		ELSIF RemoteCtrlEnable
			AND NOT RemoteDataToSlaves._WORDS[2].8 
			AND Mode <> MasterCmdMode
		THEN (* Betriebsartenwechsel ueber RemoteCtrl ein *)
			Busy := BusyIntern 								:= TRUE; 
			state 											:= eSTATE.STOPPING;
		ELSIF NOT RemoteCtrlEnable
			OR 	
			RemoteCtrlEnable
			AND MasterCmdState <> eSTATE.SUSPENDED
			AND MasterCmdState <> eSTATE.SUSPENDING
		THEN
			IF RemoteCtrlEnable 
				AND(MasterCmdState = eSTATE.UNSUSPENDING OR MasterCmdState = eSTATE.EXECUTE OR MasterCmdState = eSTATE.COMPLETING)
				OR NOT RemoteCtrlEnable
			THEN
				Busy := BusyIntern 							:= TRUE; 
				state 										:= eSTATE.UNSUSPENDING;	
			ELSE
				Busy := BusyIntern 							:= TRUE; 
				state 										:= eSTATE.STOPPING;
			END_IF
		END_IF
	{endregion} 	
	{region "UNSUSPENDING"}	
	eSTATE.UNSUSPENDING: info 								:= TO_STRING(eSTATE.UNSUSPENDING);
	
		IF GoToAborting 
		THEN
			state 											:= eSTATE.ABORTING;
			Busy := BusyIntern 								:= TRUE;

		ELSIF RemoteCtrlEnable
			AND(
			MasterCmdState = eSTATE.STOPPING
			OR (* Betriebsartenwechsel ueber RemoteCtrl ein *)
			NOT RemoteDataToSlaves._WORDS[2].8 AND Mode <> MasterCmdMode)
		THEN
			state 											:= eSTATE.STOPPING;
			Busy := BusyIntern 								:= TRUE;
		ELSIF NOT Busy 
		THEN
			Busy := BusyIntern 								:= TRUE; 
			state											:= eSTATE.EXECUTE;
		END_IF
	{endregion} 	
	{region "HOLDING"}	
	eSTATE.HOLDING:		info 								:= TO_STRING(eSTATE.HOLDING);
	
		IF GoToAborting 
		THEN
			state 											:= eSTATE.ABORTING;
			Busy := BusyIntern 								:= TRUE;

		ELSIF RemoteCtrlEnable
			AND(
			MasterCmdState = eSTATE.STOPPING
			OR (* Betriebsartenwechsel ueber RemoteCtrl ein *)
			NOT RemoteDataToSlaves._WORDS[2].8 AND Mode <> MasterCmdMode)
		THEN
			state 											:= eSTATE.STOPPING;
			Busy := BusyIntern 								:= TRUE;
		ELSIF NOT Busy 
		THEN
			state 											:= eSTATE.HELD;		
		END_IF	
	{endregion} 	
	{region "HELD"}	
	eSTATE.HELD:		info 								:= TO_STRING(eSTATE.HELD);
	
		IF GoToAborting 
		THEN
			Busy := BusyIntern 								:= TRUE; 
			state 											:= eSTATE.ABORTING;
		ELSIF RemoteCtrlEnable
			AND NOT RemoteDataToSlaves._WORDS[2].8 
			AND Mode <> MasterCmdMode
		THEN (* Betriebsartenwechsel ueber RemoteCtrl ein *)
			Busy := BusyIntern 								:= TRUE; 
			state 											:= eSTATE.STOPPING;
		ELSIF NOT RemoteCtrlEnable
			OR 	
			RemoteCtrlEnable
			AND MasterCmdState <> eSTATE.HELD
			AND MasterCmdState <> eSTATE.HOLDING
		THEN
			IF RemoteCtrlEnable 
				AND(MasterCmdState = eSTATE.EXECUTE OR MasterCmdState = eSTATE.UNHOLDING OR MasterCmdState = eSTATE.COMPLETING)
				OR NOT RemoteCtrlEnable
			THEN
				Busy := BusyIntern 							:= TRUE; 
				state 										:= eSTATE.UNHOLDING;	
			ELSE
				Busy := BusyIntern 							:= TRUE; 
				state 										:= eSTATE.STOPPING;
			END_IF
		END_IF
	{endregion} 	
	{region "UNHOLDING"}	
	eSTATE.UNHOLDING: 	info 								:= TO_STRING(eSTATE.UNHOLDING);
	
		IF GoToAborting 
		THEN
			state 											:= eSTATE.ABORTING;
			Busy := BusyIntern 								:= TRUE;

		ELSIF RemoteCtrlEnable
			AND(
			MasterCmdState = eSTATE.STOPPING
			OR (* Betriebsartenwechsel ueber RemoteCtrl ein *)
			NOT RemoteDataToSlaves._WORDS[2].8 AND Mode <> MasterCmdMode)
		THEN
			state 											:= eSTATE.STOPPING;
			Busy := BusyIntern 								:= TRUE;
		ELSIF NOT Busy 
		THEN
			Busy := BusyIntern 								:= TRUE; 
			state											:= eSTATE.EXECUTE;
		END_IF
	{endregion} 	
	{region "COMPLETING"}	
	eSTATE.COMPLETING: info 								:= TO_STRING(eSTATE.COMPLETING);
	
		IF GoToAborting 
		THEN
			Busy := BusyIntern 								:= TRUE; 
			state 											:= eSTATE.ABORTING;

		ELSIF RemoteCtrlEnable
			AND( (* Betriebsartenwechsel ueber RemoteCtrl ein *)
			MasterCmdState = eSTATE.STOPPING
			OR 
			NOT RemoteDataToSlaves._WORDS[2].8  AND Mode <> MasterCmdMode)
			OR	
			NOT RemoteCtrlEnable AND NOT Options.5 (* Cancel Completing *)
		THEN
			Busy := BusyIntern 								:= TRUE; 
			state 											:= eSTATE.STOPPING;

		ELSIF NOT Busy
		THEN
			state 											:= eSTATE.COMPLETE;
		END_IF
	{endregion} 	
	{region "COMPLETE"}	
	eSTATE.COMPLETE: info 									:= TO_STRING(eSTATE.COMPLETE);
		
		IF GoToAborting 
		THEN
			Busy := BusyIntern 								:= TRUE; 
			state 											:= eSTATE.ABORTING;

		ELSIF NOT RemoteCtrlEnable
			OR	
			RemoteCtrlEnable
			AND MasterCmdState <> eSTATE.COMPLETE
			AND MasterCmdState <> eSTATE.COMPLETING
		THEN
			Busy := BusyIntern 								:= TRUE; 
			state 											:= eSTATE.STOPPING;
		END_IF
	{endregion} 	
	{region "ABORTING"}	
	eSTATE.ABORTING: info 									:= TO_STRING(eSTATE.ABORTING);
		
		IF NOT Busy
			OR NOT EStopDelayOK
			OR RemoteCtrlEnable AND NOT MasterCmdInfo.15 (* EStop Delay False *)
		THEN
			StateComplete(); (* Ueber Hardware vorgegeben *)
			state 											:= eSTATE.ABORTED;
		END_IF
	{endregion} 	
	{region "ABORTED"}	
	eSTATE.ABORTED: info 									:= TO_STRING(eSTATE.ABORTED);
		
		IF NOT RemoteCtrlEnable AND EStopDirectOK AND EStopDelayOK
			OR 	
			RemoteCtrlEnable
			AND(EStopDirectOK AND EStopDelayOK OR Options.3)
			AND MasterCmdState <> eSTATE.ABORTED
			AND MasterCmdState <> eSTATE.ABORTING
			AND MasterCmdState <> eSTATE.STARTUP
		THEN
			Busy := BusyIntern 								:= TRUE; 
			state 											:= eSTATE.CLEARING;
		ELSE			
			(* Ack error in aborted *)
			IF LocalReset
			THEN
		 		ErrHdl.reset();
			END_IF
		END_IF
		
		(* set Mode *)
		IF Options.0
		THEN
			Mode 											:= eMODE.IDLE;
		ELSE (* take the current mode back *)
			Mode 											:= SEL(RemoteCtrlEnable,SetMode,MasterCmdMode);
		END_IF
	{endregion} 	
	{region "CLEARING"}	
	eSTATE.CLEARING: info 									:= TO_STRING(eSTATE.CLEARING);
		
		IF GoToAborting 
		THEN
			Busy := BusyIntern 								:= TRUE; 
			state 											:= eSTATE.ABORTING;
		ELSIF NOT Busy
			AND(EStopOK OR Options.3) (* Local EStop Disabled *)
			AND(MasterCmdInfo.14 OR NOT RemoteCtrlEnable) (* RemoteCtrl EStop OK *)
		THEN
			state 											:= eSTATE.STOPPED;
		END_IF
	{endregion} 	
	{region "STOPPING"}	
	eSTATE.STOPPING: Info									:= TO_STRING(eSTATE.STOPPING);
		
		IF GoToAborting 
		THEN
			Busy := BusyIntern 								:= TRUE; 
			state 											:= eSTATE.ABORTING;
		ELSIF NOT Busy 
		THEN
			state 											:= eSTATE.STOPPED;
		END_IF
	{endregion} 	
	{region "STOPPED"}	
	eSTATE.STOPPED: info 									:= TO_STRING(eSTATE.STOPPED);
		
		IF GoToAborting 
		THEN
			Busy := BusyIntern 								:= TRUE; 
			state 											:= eSTATE.ABORTING;
		ELSIF LocalReset AND ErrHdl.flag
			AND(NOT RemoteCtrlEnable OR MasterCmdState <> eSTATE.STOPPED) (* Weiter ueber Quitt im Fehlerfall *)
			AND(ErrHdl.id <> ERROR_MACHINE OR NOT Options.4)
			OR 
			NOT RemoteCtrlEnable
			AND(NOT ErrHdl.flag OR NOT Options.6 AND ErrHdl.id <> ERROR_EXTERNAL) (* Automatisch weiter wenn kein Fehler, oder ACK nicht erforderlich und Fehler nicht Extern (Quittierung erfolgt dort)*)
			OR	
			RemoteCtrlEnable (* Weiter wenn Remote Unit nicht in Stopped/Completing und nicht in Fehler *)
			AND MasterCmdState <> eSTATE.STOPPED
			AND MasterCmdState <> eSTATE.STOPPING
			AND MasterCmdState <> eSTATE.CLEARING
			AND MasterCmdState <> eSTATE.COMPLETING 
			AND MasterCmdState <> eSTATE.COMPLETE
			AND(NOT ErrHdl.flag OR NOT Options.6)
			OR 
			RemoteCtrlEnable (* Weiter wenn Maschinenfehler resetet wird *)
			AND MasterCmdState = eSTATE.RESETTING
			AND ErrHdl.flag //(MasterCmdInfo.11 or MasterCmdInfo.12 OR MasterCmdInfo.13) //OR ErrHdl.id = ERROR_MACHINE ist Bit 12)
		THEN
			Busy := BusyIntern 								:= TRUE; 
			ErrHdl.reset();
			state 											:= eSTATE.RESETTING;
		END_IF
	
		(* set Mode *)
		IF Options.0 
		THEN
			Mode 											:= eMODE.IDLE;
		ELSE (* take the current mode back *)
			Mode 											:= SEL(RemoteCtrlEnable,SetMode,MasterCmdMode);
		END_IF
	{endregion} 	
	{region "RESETTING"}	
	eSTATE.RESETTING: info 									:= TO_STRING(eSTATE.RESETTING);
		
		IF GoToAborting 
		THEN
			Busy := BusyIntern 								:= TRUE; 
			state 											:= eSTATE.ABORTING;
		ELSIF MasterCmdState = eSTATE.STOPPING 
			AND RemoteCtrlEnable 
		THEN
			Busy := BusyIntern 								:= TRUE; 
			state 											:= eSTATE.STOPPING;
		ELSIF NOT Busy 
		THEN
			state 											:= eSTATE.IDLE;
		END_IF
	{endregion} 	

	ELSE
		info 												:= CONCAT('ERROR unkown state ', TO_STRING(state));
		ErrHdl.flag 										:= TRUE;
		ErrHdl.fnc 											:= 'SubCtrl';
		ErrHdl.id											:= 99;
		ErrHdl.state										:= state;
		ErrHdl.text 										:= CONCAT('unkown state:',DINT_TO_STRING(ErrHdl.state));
		SetLocalError();
	END_CASE
		 
(* State Check *************************************************)
	RT_StateChanged 										:= LastState <> State;
	LastState 												:= State;
	
(* Statebits ***********************************************************************************)
	InStartup												:= state = eSTATE.STARTUP;
	InIdle													:= state = eSTATE.IDLE;
	InStarting												:= state = eSTATE.STARTING;
	InStarted												:= state = eSTATE.STARTED;
	InExecute												:= state = eSTATE.EXECUTE;
	InCompleting											:= state = eSTATE.COMPLETING;
	InComplete												:= state = eSTATE.COMPLETE;
	InAborting												:= state = eSTATE.ABORTING;
	InAborted												:= state = eSTATE.ABORTED;
	InClearing												:= state = eSTATE.CLEARING;
	InStopping												:= state = eSTATE.STOPPING;
	InStopped												:= state = eSTATE.STOPPED;
	InResetting												:= state = eSTATE.RESETTING;

	EStopStartupOK											:= 	NOT InAborted 
																AND(
																EStopStartupOK 
																OR 
																NOT InAborting AND NOT InClearing 
																AND NOT InStartup AND NOT InStopped );
                    										
(* optional
	InSuspending	:= state = eSTATE.SUSPENDING;
	InSuspended		:= state = eSTATE.SUSPENDED;
	InUnsuspending	:= state = eSTATE.UNSUSPENDING;

	InHolding		:= state = eSTATE.HOLDING;
	InHeld			:= state = eSTATE.HELD;
	InUnholding		:= state = eSTATE.UNHOLDING;
*)

(***************************************************************)
(* Read Subs Status and synchronize							   *)
(***************************************************************)		
{region "Check slave states and send command"}	
	(* Init Flag, all Subs in same state *)
	NoSlavesConnected										:= TRUE;
	SlavesInSync 											:= NOT RT_StateChanged;
	SlavesBusy    											:= FALSE;
	NoOfBusySlaves											:= 0;
	(* Init remote command data to slaves  *)
	RemoteDataToSlaves._INTs[0]								:= Mode;
	RemoteDataToSlaves._WORDS[2]							:= TO_WORD(Options);
	RemoteDataToSlaves._WORDS[2].8							:= RemoteCtrlEnable;
	RemoteDataToSlaves._WORDS[2].9							:= LocalReset;	
	RemoteDataToSlaves._WORDS[2].14							:= EStopOK OR Options.3;
	RemoteDataToSlaves._WORDS[2].15							:= EStopDelayOK OR Options.3;	
	RemoteDataToSlaves._INTs[3]								:= Id;
		
	(* read Subs state an send cmd to all subs *)
	FOR i := MIN_SLAVE TO MAX_SLAVE DO
		IF ipSlave[i] <> 0 
		THEN 
			NoSlavesConnected 								:= FALSE;(* pointer is used *)
			RemoteDataFromSlave								:= ipSlave[i].remoteData; //Read remote status data from slaves
			IF RemoteDataFromSlave._WORDS[2].8 
			THEN (* External Sub is Remote-Controlled *)
				(* Check the status from then external subs *)
				IF((RemoteDataFromSlave._WORDS[2].11 OR RemoteDataFromSlave._WORDS[2].13) 
					AND RemoteDataFromSlave._WORDS[2].4)(* Maschine to Remotesystem if Enabled, or External Error *)
					AND NOT ErrHdl.flag
					AND NOT InStartup AND NOT InResetting
					AND NOT InAborting AND NOT InAborted
				THEN (* external sub has fatal error *)
					(* external subs send fatal machine error -> bring local sub in Stopping with error *)
					ErrHdl.flag								:= TRUE;
					ErrHdl.state							:= state;
					ErrHdl.fnc 								:= name;
					ErrHdl.id								:= ERROR_EXTERNAL;
					ErrHdl.text 							:= CONCAT('Fatal machine error in Sub index no.:',INT_TO_STRING(i));
					Busy									:= state <> eSTATE.STOPPING;
					state 									:= eSTATE.STOPPING;
					SlavesInSync 							:= FALSE;
				ELSE (* external sub has no error *)
					IF SlavesState = RemoteDataFromSlave._INTs[1]
					THEN (* Check if sub is in sync with other subs *)
						SlavesState 						:= RemoteDataFromSlave._INTs[1];
					ELSE (* external sub is not in sync with other subs *)
						IF (RemoteDataFromSlave._INTs[1] = eSTATE.ABORTED OR RemoteDataFromSlave._INTs[1] = eSTATE.ABORTING)
							AND NOT InAborted 
							AND NOT InAborting
							AND NOT RemoteDataFromSlave._WORDS[2].3 (* Local EStop-Signals Disable *)
							OR RemoteDataFromSlave._WORDS[2].11 (* Maschine Error *)
							OR RemoteDataFromSlave._WORDS[2].12 (* Local Error  *)
							OR RemoteDataFromSlave._WORDS[2].13 (* External Error  *)
							OR (* comleting at sub disabled *)
							NOT RemoteDataFromSlave._WORDS[2].5 
							AND(InCompleting OR InComplete)
							AND(RemoteDataFromSlave._INTs[1] = eSTATE.STOPPING OR RemoteDataFromSlave._INTs[1] = eSTATE.STOPPED)
						THEN
							; (* ignore cause sub use local EStop-signals, or error in stopped *)
						ELSE
							SlavesState						:= RemoteDataFromSlave._INTs[2];
							SlavesInSync 					:= FALSE;
						END_IF
					END_IF

					(* subs busy *)
					IF (RemoteDataFromSlave._INTs[1] = eSTATE.ABORTED OR RemoteDataFromSlave._INTs[1] = eSTATE.ABORTING )
						AND NOT InAborted 
						AND NOT InAborting
						AND NOT RemoteDataFromSlave._WORDS[2].3 (* Local EStop-Signals Disable *)
						OR RemoteDataFromSlave._WORDS[2].12 (* Local Error *)
						OR 
						SlavesState = eSTATE.EXECUTE AND NOT InExecute
					THEN
						; (* ignore cause sub is in error or use local EStop-Signals *)
					ELSIF RemoteDataFromSlave._WORDS[2].10 
					THEN
						SlavesBusy 							:= TRUE;
						NoOfBusySlaves						:= NoOfBusySlaves + 1;
					END_IF

				END_IF
			ELSE (* external Sub is not in RemoteCtrl *)
				;
			END_IF

			(* Write latest command data   *)
			RemoteDataToSlaves._INTs[1]						:= State;
			RemoteDataToSlaves._WORDS[2].10					:= Busy;
			RemoteDataToSlaves._WORDS[2].11					:= ErrHdl.id = ERROR_MACHINE;
			RemoteDataToSlaves._WORDS[2].12					:= ErrHdl.id = ERROR_LOCAL;
			RemoteDataToSlaves._WORDS[2].13					:= ErrHdl.id = ERROR_EXTERNAL;

			(* set slave command data *)
			ipSlave[i].remoteData							:= RemoteDataToSlaves; //Write data as command to every slave
		ELSE
			EXIT; (* pointer not used -> Exit for *)
		END_IF
	END_FOR

	(* Set state complete only if all Subs in the same state or current state is Execute *)
	IF SlavesInSync AND NOT NoSlavesConnected 
	THEN //Subs in sync
		IF SlavesBusy 
			OR (BusyIntern AND Options.2) 
			OR (NOT EStopOK AND NOT Options.3 AND InClearing) (* Solange Busy halten, biss durch EStopOK aus Clearing gegangen werden kann *)
		THEN
			; (* al least one sub is busy or not StateComplete *)
		ELSIF Busy 
		THEN
			Busy := BusyIntern 								:= FALSE; (* All subs not StateComplete (NOT Busy) set UnitSub StateComplete *)
		END_IF
	END_IF
{endregion}
	 
(* Set Status RemoteData for master to check ************************************************************)
	RemoteDataToSlaves._INTs[0] 							:= Mode;
	RemoteDataToSlaves._INTs[1]								:= State;
	RemoteDataToSlaves._WORDs[2]							:= TO_WORD(Options);
	RemoteDataToSlaves._WORDs[2].8							:= RemoteCtrlEnable;
	RemoteDataToSlaves._WORDs[2].9							:= LocalReset;
	RemoteDataToSlaves._WORDs[2].10							:= Busy;
	RemoteDataToSlaves._WORDs[2].11							:= ErrHdl.id = ERROR_MACHINE;
	RemoteDataToSlaves._WORDs[2].12							:= ErrHdl.id = ERROR_LOCAL;
	RemoteDataToSlaves._WORDs[2].13							:= ErrHdl.id = ERROR_EXTERNAL;
	RemoteDataToSlaves._WORDs[2].14							:= EStopOK OR Options.3;
	RemoteDataToSlaves._WORDs[2].15							:= EStopDelayOK OR Options.3;
	RemoteDataToSlaves._INTs[3]								:= Id;
	

(* Reset LocalAck ******************************************************************************)
	Localreset												:= FALSE;

(***********************************************************************************************)

METHOD PRIVATE FINAL _createID : INT
VAR_STAT //Value is stored for each instance
	IdCnt													: INT;
END_VAR
IdCnt														:= IdCnt + 1;
_CreateID 													:= IdCnt;
END_METHOD

METHOD PUBLIC FINAL addSlave : BOOL
VAR_INPUT
	ipSlave													:	I_Statemodel;
END_VAR
addSlave													:= FALSE;	
IF ipSlave <> 0	
then
	FOR i := MIN_SLAVE TO MAX_SLAVE
	DO 
		IF ipSlave = THIS^.ipSlave[i] THEN
			addSlave										:= TRUE;
			EXIT;
		ELSIF THIS^.ipSlave[i] = 0
		THEN								
			THIS^.ipSlave[i]								:= ipSlave;
			addSlave										:= TRUE;
			EXIT;
		END_IF
	END_FOR
END_IF
END_METHOD

METHOD FB_init : BOOL
VAR_INPUT
	bInitRetains : BOOL; // if TRUE, the retain variables are initialized (warm start / cold start)
	bInCopyCode : BOOL;  // if TRUE, the instance afterwards gets moved into the copy code (online change)
END_VAR
(* Generate ID ****************************************************)
	IF Id = 0 
	THEN 
		id 													:= _CreateID(); 
		IF Name = '' 
		THEN 
			Name 											:= CONCAT('Statemodel Id ',TO_STRING(Id)); 
		ELSE
			Name 											:= CONCAT(Name , CONCAT(' Id ', TO_STRING(Id))); 
		END_IF
	END_IF	
(***********************************************************************)
END_METHOD

METHOD PUBLIC isModeActive : BOOL
VAR_INPUT
	Mode													: eMODE;				
END_VAR
IsModeActive := Mode = THIS^.Mode AND(InExecute OR InCompleting);
END_METHOD

METHOD PUBLIC isStateActive : BOOL
VAR_INPUT
	state								: eSTATE;
END_VAR
IsStateActive := state = This^.State;
END_METHOD

METHOD PUBLIC reset : boOL //Result = TRUE if Resetting finished - ErrHdl.Flag = FALSE
VAR_INPUT
END_VAR
LocalReset													:= TRUE;
reset														:= NOT ErrHdl.flag;
END_METHOD

METHOD PUBLIC setLocalError : booL
VAR_INPUT
END_VAR
IF NOT ErrHdl.flag
	AND state <> eSTATE.ABORTING
	AND state <> eSTATE.ABORTED
	AND state <> eSTATE.CLEARING
	and state <> eSTATE.RESETTING
THEN
	ErrHdl.flag 											:= TRUE;
	ErrHdl.state											:= state;
	ErrHdl.fnc												:= name;
	ErrHdl.id												:= ERROR_LOCAL;
	ErrHdl.text 											:= 'Local ctrl error';
	Busy													:= state <> eSTATE.STOPPING;
	state 													:= eSTATE.STOPPING;
	SetLocalError											:= TRUE;
ELSE
	SetLocalError											:= ErrHdl.id = ERROR_LOCAL;
END_IF
END_METHOD

METHOD PUBLIC setMachineError : booL
VAR_INPUT
END_VAR
IF NOT ErrHdl.flag
	AND state <> eSTATE.ABORTING
	AND state <> eSTATE.ABORTED
	AND state <> eSTATE.CLEARING
	AND state <> eSTATE.RESETTING
THEN
	ErrHdl.flag												:= TRUE;
	ErrHdl.state											:= state;
	ErrHdl.fnc												:= name;
	ErrHdl.id												:= ERROR_MACHINE;
	ErrHdl.text 											:= 'Fatal machine error';
	Busy													:= state <> eSTATE.STOPPING;
	state 													:= eSTATE.STOPPING;
	SetMachineError											:= TRUE;
ELSE
	SetMachineError											:= ErrHdl.id = ERROR_MACHINE;;
END_IF
END_METHOD

METHOD PUBLIC FINAL stateComplete : BOOL //Result = TRUE if state completed (BusyIntern=FALSE)
VAR_INPUT
END_VAR
BusyIntern 													:= FALSE;
StateComplete												:= NOT BusyIntern AND NOT Busy;
END_METHOD

{attribute 'monitoring' := 'call'}
PROPERTY PUBLIC optDisableSafetyInputs : BOOL
GET
optDisableSafetyInputs := Options.3;
END_GET
SET
Options.3 := optDisableSafetyInputs;
END_SET
END_PROPERTY

{attribute 'monitoring' := 'call'}
PROPERTY PUBLIC optEnableAutoChangeModeToIdle : BOOL
GET
optEnableAutoChangeModeToIdle := Options.0;
END_GET
SET
Options.0 := optEnableAutoChangeModeToIdle;
END_SET
END_PROPERTY

{attribute 'monitoring' := 'call'}
PROPERTY PUBLIC optEnableExplicitReset : BOOL
GET
optEnableExplicitReset := Options.6;
END_GET
SET
Options.6 := optEnableExplicitReset;
END_SET
END_PROPERTY

{attribute 'monitoring' := 'call'}
PROPERTY PUBLIC optEnableExternalStateComplete : BOOL
GET
optEnableExternalStateComplete := Options.2;
END_GET
SET
Options.2 := optEnableExternalStateComplete;
END_SET
END_PROPERTY

{attribute 'monitoring' := 'call'}
PROPERTY PUBLIC optEnableFwdMachineErrorToMaster : BOOL
GET
optEnableFwdMachineErrorToMaster := Options.4;
END_GET
SET
Options.4 := optEnableFwdMachineErrorToMaster;
END_SET
END_PROPERTY

{attribute 'monitoring' := 'call'}
PROPERTY PUBLIC optEnableModeChangeInExecute : BOOL
GET
optEnableModeChangeInExecute := Options.1;
END_GET
SET
Options.1 := optEnableModeChangeInExecute;
END_SET
END_PROPERTY

{attribute 'monitoring' := 'call'}
PROPERTY PUBLIC optEnableModeChangeViaStateCompl : BOOL
GET
optEnableModeChangeViaStateCompl := Options.5;
END_GET
SET
Options.5 := optEnableModeChangeViaStateCompl;
END_SET
END_PROPERTY

{attribute 'monitoring' := 'call'}
PROPERTY public actMode : eMODE
GET
actMode := Mode;
END_GET
END_PROPERTY

{attribute 'monitoring' := 'call'}
PROPERTY public actState : eSTATE
GET
actState := state;
END_GET
END_PROPERTY

{attribute 'monitoring' := 'call'}
PROPERTY PUBLIC ipMasterUnit : I_Statemodel //The slave will add his interface pointer into the master through this propertiy
SET
IF IdRemoteMaster = 0 AND_THEN ipMasterUnit <> 0
THEN
	RemoteDataToSlaves									:= ipMasterUnit.remoteData;	
	IF IdRemoteMaster <> RemoteDataToSlaves._INTs[3] 
	THEN
		IF ipMasterUnit.addSlave(THIS^)
		THEN					
			remoteData 									:= RemoteDataToSlaves; 
		END_IF
	END_IF
END_IF
END_SET
END_PROPERTY

{attribute 'monitoring' := 'call'}
PROPERTY isBusy : BOOL
GET
isBusy := Busy;
END_GET
END_PROPERTY

PROPERTY public remoteData : U_64BIT_DATATYPE
GET
//statis of sub
remoteData := RemoteDataToSlaves;
END_GET
SET
//Cmd to sub
MasterCmdMode 	:= remoteData._INTs[0];
MasterCmdState := remoteData._INTs[1];
MasterCmdInfo 	:= remoteData._WORDS[2];
IdRemoteMaster := remoteData._INts[3];
END_SET
END_PROPERTY

{attribute 'monitoring' := 'call'}
PROPERTY PUBLIC rErrHdl : REFERENCE to ERROR_HDL
GET
rErrHdl REF= Errhdl;
END_GET
END_PROPERTY

PROPERTY PUBLIC setStateComplete : BOOL
GET
SetStateComplete := not BusyIntern and not Busy;
END_GET
SET
IF SetStateComplete AND BusyIntern
THEN
	StateComplete();
END_IF
END_SET
END_PROPERTY

END_FUNCTION_BLOCK

// POUs/Statemodel/control/I_Statemodel
INTERFACE I_Statemodel extends I_StatemodelBase

METHOD PUBLIC FINAL addSlave : BOOL
VAR_INPUT
	ipSlave					:	I_Statemodel;
END_VAR
END_METHOD

METHOD PUBLIC isModeActive : BOOL
VAR_INPUT
	Mode													: eMODE;				
END_VAR
END_METHOD

METHOD PUBLIC isStateActive : BOOL
VAR_INPUT
	state						:	eSTATE;
END_VAR
END_METHOD

METHOD PUBLIC reset : boOL //Result = TRUE if Resetting finished - ErrHdl.Flag = FALSE
VAR_INPUT
END_VAR
END_METHOD

METHOD PUBLIC setLocalError : booL
VAR_INPUT
END_VAR
END_METHOD

PROPERTY public remoteData : U_64BIT_DATATYPE
GET
END_GET
SET
END_SET
END_PROPERTY

{attribute 'monitoring' := 'call'}
PROPERTY PUBLIC rErrHdl : REFERENCE to ERROR_HDL
GET
END_GET
END_PROPERTY

END_INTERFACE

// POUs/Statemodel/control/I_StatemodelBase
INTERFACE I_StatemodelBase Extends __System.IQueryInterface

METHOD PUBLIC setMachineError : booL
VAR_INPUT
END_VAR
END_METHOD

METHOD PUBLIC stateComplete : BOOL //Result = TRUE if state completed (BusyIntern=TRUE)
VAR_INPUT
END_VAR
END_METHOD

{attribute 'monitoring' := 'call'}
PROPERTY public actMode : eMODE
GET
END_GET
END_PROPERTY

{attribute 'monitoring' := 'call'}
PROPERTY public actState : eSTATE
GET
END_GET
END_PROPERTY

{attribute 'monitoring' := 'call'}
PROPERTY isBusy : BOOL
GET
END_GET
END_PROPERTY

PROPERTY PUBLIC setStateComplete : BOOL
GET
END_GET
SET
END_SET
END_PROPERTY

END_INTERFACE

// POUs/Statemodel/UnitTemplate/Statemodel_Unit
{attribute 'no_check'}
//Generic Unit 
FUNCTION_BLOCK Statemodel_Unit implements I_Statemodel_Unit
VAR_OUTPUT CONSTANT
END_VAR             										
VAR_INPUT           										
	unit																:	Statemodel;		
END_VAR             										
VAR_OUTPUT          										
END_VAR             	
VAR                 	
(* Local variables ************************************************************)

(* Trigger *****************************************************************)

(* Timer ******************************************************************)

(* Fcuntion blocks ***************************************************************)

(* Dummys **********************************************************)

END_VAR

	(* Generic unit incl. state model										V1.0		*)
	(************************************************************************************)

(* work local sub ****************************************)
	Unit();
	IF Unit.RT_StateChanged THEN stateChanged(unit.Mode, Unit.State); END_IF
	
(* call methods ********************************************)
	CASE Unit.state OF
	eSTATE.STARTUP			:	Startup();
	eSTATE.IDLE				: 	Idle();
	eSTATE.STARTING			:	Starting();		
	eSTATE.STARTED			: 	Started();	
	eSTATE.EXECUTE			:	Executing();
	eSTATE.COMPLETING		:	Completing();
	eSTATE.COMPLETE			: 	Complete();
	eSTATE.ABORTING			:	Aborting();
	eSTATE.ABORTED			:  	Aborted();
	eSTATE.CLEARING			:	Clearing();
	eSTATE.STOPPING			:	Stopping();
	eSTATE.STOPPED			: 	Stopped();
	eSTATE.RESETTING		:	Resetting();
	ELSE
		;
	END_CASE

(*********************************************************)

METHOD PROTECTED aborted : BOOL
VAR_INPUT
END_VAR
Aborted														:= unit.InAborted;
END_METHOD

METHOD PROTECTED aborting : BOOL
VAR_INPUT
END_VAR
Unit.StateComplete();
Aborting													:= Unit.InAborting;
END_METHOD

METHOD PROTECTED clearing : Bool
VAR_INPUT
END_VAR
Unit.StateComplete();
Clearing													:= Unit.InClearing;
END_METHOD

METHOD PROTECTED complete : Bool
VAR_INPUT
END_VAR
Complete														:= unit.InComplete;
END_METHOD

METHOD PROTECTED completing : BOOL
VAR_INPUT
END_VAR
Unit.StateComplete();
Completing													:= Unit.InCompleting;
END_METHOD

METHOD PROTECTED executing : booL
VAR_INPUT
END_VAR
Executing 												:= Unit.InExecute;
END_METHOD

METHOD FB_exit : BOOL
VAR_INPUT
	bInCopyCode : BOOL; // if TRUE, the exit method is called for exiting an instance that is copied afterwards (online change).
END_VAR
FB_EXit															:= TRUE;
END_METHOD

METHOD FB_init : BOOL
VAR_INPUT
	bInitRetains : BOOL; // if TRUE, the retain variables are initialized (warm start / cold start)
	bInCopyCode : BOOL;  // if TRUE, the instance afterwards gets moved into the copy code (online change)
END_VAR
(* Example 
	Unit.pSubRemoteData[1]												:= ADR(Infeed.unit.RemoteData);
	Unit.pSubRemoteData[2]												:= ADR(Support_1.unit.RemoteData);
	Unit.pSubRemoteData[3]												:= ADR(Support_2.RemoteData);	
	Unit.pSubRemoteData[4]												:= ADR(Transport.unit.RemoteData);
	Unit.pSubRemoteData[5]												:= ADR(Outfeed.unit.RemoteData);
*)
FB_init														:= TRUE;
END_METHOD

METHOD FB_reinit : BOOL
VAR_INPUT
END_VAR
FB_reinit											:= TRUE;
END_METHOD

METHOD PROTECTED idle : Bool
VAR_INPUT
END_VAR
Idle														:= unit.InIdle;
END_METHOD

METHOD PROTECTED Resetting : Bool
VAR_INPUT
END_VAR
Unit.StateComplete();
Resetting													:= Unit.InResetting;
END_METHOD

{attribute 'monitoring' := 'call'}
PROPERTY public rUnit : REFERENCE TO Statemodel
GET
rUnit REF= Unit;
END_GET
END_PROPERTY

METHOD PROTECTED started : Bool
VAR_INPUT
END_VAR
Started													:= Unit.InStarted;
END_METHOD

METHOD PROTECTED starting : Bool
VAR_INPUT
END_VAR
Unit.StateComplete();
Starting													:= Unit.InStarting;
END_METHOD

METHOD PROTECTED startup : Bool
VAR_INPUT
END_VAR
Unit.StateComplete();
Startup													:= Unit.InStartup;
END_METHOD

METHOD PROTECTED stateChanged : BOOL 
VAR_INPUT
	mode											:	eMODE;
	state											:	eSTATE;
END_VAR
END_METHOD

METHOD PROTECTED stopped : Bool
VAR_INPUT
END_VAR
Stopped														:= unit.InStopped;
END_METHOD

METHOD PROTECTED stopping : Bool
VAR_INPUT
END_VAR
Unit.StateComplete();
Stopping													:= Unit.InStopping;
END_METHOD

END_FUNCTION_BLOCK

// POUs/Statemodel/UnitTemplate/I_Statemodel_Unit
INTERFACE I_Statemodel_Unit Extends __System.IQueryInterface

{attribute 'monitoring' := 'call'}
PROPERTY public rUnit : REFERENCE TO Statemodel
GET
END_GET
END_PROPERTY

END_INTERFACE

// POUs/Motion/TF50xx-NC/03_Utilities/CoordinateTransformation2D
FUNCTION_BLOCK CoordinateTransformation2D //CoordinateTransformation
// transformation of an X/Y product coordinate to the machine coordinate system
// MCS = machine coordinate system
// PCS = product coordinate system
VAR_INPUT
//Parameter
	x0 														: LREAL;		// origin MCS X coordinate of the product coordinate system
	y0 														: LREAL;		// origin MCS Y coordinate of the product coordinate system
	x1 														: LREAL;		// opposite corner point MCS X coordinate of the product 
	y1 														: LREAL;		// opposite corner point MCS Y coordinate of the product
	a 														: LREAL;		// length of the product (difference x1pcs-x0pcs)
	b 														: LREAL;		// width of the product (difference y1pcs-y0pcs)
END_VAR                                                 	
VAR_OUTPUT                                              	
	Xmcs 													: LREAL;	// X coordinate in machine coordinate system
	Ymcs 													: LREAL;	// Y coordinate in machine coordinate system
															
	Xpcs 													: LREAL;	// X coordinate in Product coordinate system
	Ypcs 													: LREAL;	// Y coordinate in Product coordinate system
                                                        	
	Alfa													: LREAL;	

	Error 													: BOOL;	
//		ErrorID 											: UDINT;
END_VAR
VAR
	c														: LREAL;
	diagonal												: LREAL;

	ratio													: LREAL;
	
	alfa1													: LREAL;
	alfa2													: LREAL;
END_VAR

;

{attribute 'monitoring' := 'call'}
PROPERTY PUBLIC diagonalMSC : LREAL
GET
VAR
	t		:	LREAL;
END_VAR
t 			:=  EXPT(X1-X0,2.0) + EXPT(y1-y0,2.0);
DiagonalMSC := SQRT(t);
END_GET
END_PROPERTY

{attribute 'monitoring' := 'call'}
PROPERTY PUBLIC diagonalPCS : LREAL
GET
DiagonalPCS := SQRT((a*a)+(b*b));
END_GET
END_PROPERTY

{attribute 'monitoring' := 'call'}
PROPERTY PUBLIC isParamValid : BOOL
GET
IsParamValid 													:= not ParamHasError;
END_GET
SET
PUBLIC 
VAR
END_VAR
IF NOT IsParamValid
THEN
	a 														:= 0.0;
	b 														:= 0.0;
	x1 														:= Y1 := 0.0;
	y0 														:= X0 := 0.0;
END_IF
END_SET
END_PROPERTY

METHOD MSCtoPCS : BOOL //Return value = TRUE if execution finished successful / FALSE if finished with error
VAR_INPUT
	Xmcs 													: LREAL;	// X coordinate in machine coordinate system
	Ymcs 													: LREAL;	// Y coordinate in machine coordinate system
END_VAR
IF ParamHasError THEN
	Error 													:= TRUE; 
	MSCtoPCS 												:= FALSE;
ELSE	
	THIS^.Xmcs												:= Xmcs;	
	THIS^.Ymcs												:= Ymcs;	

	c 														:= SQRT(a*a + b*b);
	alfa 													:= ACOS((x1-x0) / c) - ACOS( a / c);
	
	Xpcs 													:= 	 (Xmcs - x0) * COS(alfa) + (Ymcs - y0) * SIN(alfa);
	Ypcs 													:= - (Xmcs - x0) * SIN(alfa) + (Ymcs - y0) * COS(alfa);
	
	Error 													:= FALSE; 
	MSCtoPCS 												:= TRUE;
END_IF
END_METHOD

{attribute 'monitoring' := 'call'}
PROPERTY PRIVATE paramHasError : BOOL
GET
ParamHasError := 	a<=0.0 
			OR 	b<=0.0 
			OR 	x1=x0 
			OR 	y1=y0;
END_GET
END_PROPERTY

METHOD PUBLIC PCStoMSC : booL //Return value = TRUE if execution finished successful / FALSE if finished with error
VAR_INPUT
	Xpcs : LREAL;	// X coordinate in product coordinate system
	Ypcs : LREAL;	// Y coordinate in product coordinate system	
END_VAR
IF ParamHasError 
THEN
	Error 													:= TRUE; 
	PCStoMSC												:= FALSE;
ELSE                										
	THIS^.Xpcs												:= Xpcs;	
	THIS^.Ypcs												:= Ypcs;
	
	c 														:= SQRT(a*a + b*b);
	diagonal												:= SQRT((x1-x0)*(x1-x0)+(y1-y0)*(y1-y0));
	
	ratio													:= diagonal/c;
	
	alfa1 													:= ACOS((x1-x0) / diagonal);
	alfa2													:= ACOS(a/c);
	
	alfa													:= alfa1-alfa2;
	
	Xmcs 													:= x0 + ratio * (Xpcs * COS(alfa) - Ypcs * SIN(alfa));
	Ymcs 													:= y0 + ratio * (Xpcs * SIN(alfa) + Ypcs * COS(alfa));
                    	
	Error 													:= FALSE; 
	PCStoMSC												:= TRUE;
END_IF
END_METHOD

END_FUNCTION_BLOCK

// POUs/Motion/TF50xx-NC/03_Utilities/getOvrVelo
{attribute 'no_check'}
//Overwrite function - Returns velocity setpoint based on max velo and requested overwrite 
FUNCTION getOvrVelo : LREAL
VAR_INPUT
	SetVelo													:	LREAL;
	MaxVelo													:	LREAL;
END_VAR
VAR
END_VAR

IF 	MaxVelo = 0.0 OR SetVelo = 0.0
THEN
	GetOvrVelo 												:= 0.0;
ELSE                										
	GetOvrVelo 												:= 100.0 / MaxVelo * SetVelo;
END_IF

END_FUNCTION

// POUs/Motion/TF50xx-NC/AxNcBase
FUNCTION_BLOCK AxNcBase EXTENDS AXIS_REF IMPLEMENTS I_AxNcBase(* See Tc2_MC2 *)
VAR_OUTPUT CONSTANT
	OPTION_EN_CMD_ABORTED_ERROR								: 	BYTE := 2#1000_0000; //Default: .7 = xxx.CmdAborted is treaded as error
END_VAR
VAR_INPUT
{attribute 'displaymode':='binary'}
	Options													: 	BYTE  := OPTION_EN_CMD_ABORTED_ERROR; //See output constant for Options mask
	
(* Axis *)
	Admin													: 	AxAdmin;
	para													: 	AxPara;

	Home													:	AxHoming;
	event													:	AxEventHandling;                                                   
END_VAR                                             	
VAR_OUTPUT                                          	
	ErrHdl													:	ERROR_HDL;
END_VAR
VAR
END_VAR

	(* Axis 																*)
	(************************************************************************)

	
(********************************************************************************)
(* Error NC																		*)
(********************************************************************************)
	Event(
		Enable		:= Admin.EnableOK OR Event.NoOfActiveEvents > 0,
		ConfirmTrig	:= Admin.ResetTrig,
		Name		:= para.Name,
		SourceId	:= (* Default *) ,
		rAxis		:= THIS^,
		ErrorId		:= TO_UDINT(ErrHdl.Id),
		Status		=> );
		
	(* Init ErrHdl *)
	ErrHdl.Reset();

(********************************************************************************)
(* work Admin ctrl 																*)
(********************************************************************************)
	Admin(rAxis		:= THIS^);
	IF Admin.Error
	THEN
		ErrHdl.id 											:= UDINT_TO_DINT(Admin.ErrorId);
		ErrHdl.fnc											:= 'Admin';
		ErrHdl.text											:= Admin.ErrorText;
		ErrHdl.flag											:= TRUE;
	END_IF
	
(********************************************************************************)
(* Parameter																	*)
(********************************************************************************)
	para(Axisid := NcToPlc.AxisId);
		
(********************************************************************************)
(* work homing ctrl 															*)
(********************************************************************************)
	Home(rAxis := THIS^ );
	errorCheck(AxBase := Home);
	

(********************************************************************************)

METHOD PROTECTED errorCheck : BOOL
VAR_IN_OUT
	AxBase									:	AxFbBase;
END_VAR
IF AxBase.Error
THEN
	ErrHdl.flag									:= TRUE;
	ErrHdl.fnc									:= 'AxNcPtP';
	ErrHdl.id									:= TO_DINT(AxBase.ErrorID);
	ErrHdl.text									:= AxBase.ErrorText;
	errorCheck									:= TRUE;
ELSIF AxBase.CmdAborted AND Options.7
THEN
	ErrHdl.id 									:= 19200;
	ErrHdl.fnc									:= 'AxNcPtP';
	ErrHdl.text									:= 'command aborted';
	ErrHdl.flag									:= TRUE;		
ELSE
	errorCheck									:= FALSE;
END_IF
END_METHOD

METHOD PUBLIC noAction : BOOL //Return value = TRUE if busy of home and motion 
VAR_INPUT
END_VAR
home.Execute	:= FALSE;


NoAction 		:= 	NOT home.Busy ;
END_METHOD

PROPERTY PUBLIC optEnableCmdAbortedAsError : BOOL
GET
optEnableCmdAbortedAsError := Options.7;
END_GET
SET
Options.7 := optEnableCmdAbortedAsError;
END_SET
END_PROPERTY

{attribute 'monitoring' := 'call'}
PROPERTY rAdmin : REFERENCE to AxAdmin
GET
rAdmin REF= Admin;
END_GET
END_PROPERTY

{attribute 'monitoring' := 'call'}
PROPERTY rAxisRef : REFERENCE TO AXIS_REF
GET
rAxisRef REF= THIS^;
END_GET
END_PROPERTY

{attribute 'monitoring' := 'call'}
PROPERTY PUBLIC rErrHdl : REFERENCE to ERROR_HDL
GET
rErrHdl REF= ErrHdl;
END_GET
SET
ErrHdl := rErrHdl;
END_SET
END_PROPERTY

METHOD reset : Bool
VAR_INPUT
END_VAR
NoAction();
reset 			:= ErrHdl.flag OR Admin.reset(FALSE);
Event.confirm();
END_METHOD

{attribute 'monitoring' := 'call'}
PROPERTY rHome : REFERENCE To AxHoming
GET
rHome REF= Home;
END_GET
END_PROPERTY

{attribute 'monitoring' := 'call'}
PROPERTY rPara : REFERENCE TO AxPara
GET
rPara REF= Para;
END_GET
END_PROPERTY

END_FUNCTION_BLOCK

// POUs/Motion/TF50xx-NC/AxNcPTP
FUNCTION_BLOCK AxNcPTP EXTENDS AxNcBase implements I_AxNcPTP (* See Tc2_MC2 *)
VAR_OUTPUT CONSTANT
END_VAR
VAR_INPUT
	Motion													:	AxMotion;                                        
END_VAR                           
VAR_OUTPUT                  	
END_VAR
VAR

END_VAR

	(* Axis 																*)
	(************************************************************************)

	
(********************************************************************************)
(* Call AxNcBase																*)
(********************************************************************************)
	Super^();
		
(********************************************************************************)
(* work moving ctrl 															*)
(********************************************************************************)
	Motion(rAxis := THIS^);
	errorCheck(AxBase := Motion);
	
(********************************************************************************)

METHOD PUBLIC noAction : BOOL //Return value = TRUE if busy of home and motion 
VAR_INPUT
END_VAR

Motion.Execute	:= FALSE;
Motion.JogBwd	:= FALSE;
Motion.JogFwd	:= FALSE;

NoAction 		:= 	Super^.noAction() and NOT Motion.Busy;
END_METHOD

{attribute 'monitoring' := 'call'}
PROPERTY rMotion : REFERENCE TO AxMotion
GET
rMotion REF= Motion;
END_GET
END_PROPERTY

END_FUNCTION_BLOCK

// POUs/Motion/TF50xx-NC/AxNcBaseExt
FUNCTION_BLOCK AxNcBaseExt EXTENDS AxNcBase 
VAR_OUTPUT CONSTANT
END_VAR
VAR_INPUT
	State													:	AxStatemodel;                                               
END_VAR                                             	
VAR_OUTPUT                                          	
END_VAR
VAR
END_VAR

	(* Axis 																*)
	(************************************************************************)

	
(********************************************************************************)
(* Call super 																	*)
(********************************************************************************)
	SUPER^();

(********************************************************************************)
(* Execute unit state model														*)
(********************************************************************************)
	State(
		Unit						:=  ,
		rAxis						:= THIS^,
		PT_DelEStopDisableAx		:= ,
		SafetyOK					:= ,//NOT Drive.SafetyError,
		ErrorActive					:= Event.ErrorId <> 0);

	//Execute aller Bausteine zuruecknehmen
	IF state.unit.InResetting 
		AND State.unit.RT_StateChanged
	THEN
		NoAction();
	END_IF

(********************************************************************************)

END_FUNCTION_BLOCK

// POUs/Motion/TF50xx-NC/AxNcPtpGear
FUNCTION_BLOCK AxNcPtpGear EXTENDS AxNcPTP
VAR_OUTPUT CONSTANT
END_VAR
VAR_INPUT
(* Axis *)
	Gear													:	AxGear;                                                
END_VAR                                             	
VAR_OUTPUT                                          	
END_VAR
VAR
END_VAR

	(* Axis extended (Incl. Gearing)										*)
	(************************************************************************)
	
(********************************************************************************)
(* work basic	 																*)
(********************************************************************************)
	SUPER^();

(********************************************************************************)
(* work gear ctrl 																*)
(********************************************************************************)
	gear(rAxis := THIS^);
	errorCheck(AxBase := Gear);
	
(********************************************************************************)

METHOD PUBLIC noAction : BOOL //Return value = TRUE if busy of home and motion 
VAR_INPUT
END_VAR
Gear.Execute	:= FALSE;

NoAction 		:= 	SUPER^.NoAction() AND NOT Gear.Busy ;
END_METHOD

METHOD reset : Bool
VAR_INPUT
END_VAR
Gear.Execute		:= FALSE;
reset 				:= SUPER^.reset();
END_METHOD

END_FUNCTION_BLOCK

// POUs/Motion/TF50xx-NC/AxNcPTPwJobs
FUNCTION_BLOCK AxNcPTPwJobs EXTENDS AxNcPTP (* See Tc2_MC2 *)
VAR_OUTPUT CONSTANT
	MIN_JOB													:	INT := 0;
	MAX_JOB													:	INT := 5;
	
{attribute 'displaymode':='binary'}
	OPTION_EN_CYCLIC_TARGET_CHECK							: 	BYTE := 2#0000_0001; //.0 = Cyclic target check	
END_VAR
VAR_INPUT
	Job														:	ARRAY[MIN_JOB..MAX_JOB] OF AX_JOB;	                              
END_VAR                           
var_output                  	
	JobId													:	INT := MIN_JOB;
END_VAR
VAR
	i 														: 	INT;
END_VAR

	(* Axis 																*)
	(************************************************************************)

	
(********************************************************************************)
(* Call AxNcBase																*)
(********************************************************************************)
	Super^();
			
(* Check start arr pos **********************************************************)
	IF Options.0 AND Para.InitDone THEN	CheckTargetPos(); END_IF
	
(********************************************************************************)

METHOD PUBLIC checkTargetPos : INT //ID of last job which is in target / 0 if no job is in target
VAR_INPUT
END_VAR
CheckTargetPos				:= 0;
FOR i := MIN_JOB TO MAX_JOB DO
	IF Job[i].Fnc = 6 THEN
		Job[i].InTarget := Status.NotMoving
									AND(
									NcToPlc.ModuloActPos >= Job[i].Target - para.TargetPosWindow
									AND NcToPlc.ModuloActPos <= Job[i].Target + para.TargetPosWindow
									OR
									(MODABS(Job[i].Target,para.ModuloFactor) <= 0 + para.TargetPosWindow
									OR MODABS(Job[i].Target,para.ModuloFactor) >= para.ModuloFactor - para.TargetPosWindow)
									AND(
									NcToPlc.ModuloActPos >= para.ModuloFactor - para.TargetPosWindow
									OR NcToPlc.ModuloActPos <= 0 + para.TargetPosWindow));

		Job[i].InPosWindow	:= NcToPlc.ModuloActPos >= Job[i].Target - para.PosRangeWindow
									AND NcToPlc.ModuloActPos <= Job[i].Target + para.PosRangeWindow
									OR
									(MODABS(Job[i].Target,para.ModuloFactor) <= 0 + para.PosRangeWindow
									OR MODABS(Job[i].Target,para.ModuloFactor) >= para.ModuloFactor - para.PosRangeWindow)
									AND(
									NcToPlc.ModuloActPos >= para.ModuloFactor - para.PosRangeWindow
									OR NcToPlc.ModuloActPos <= 0 + para.PosRangeWindow);
	ELSE
		Job[i].InTarget := Status.NotMoving
									AND NcToPlc.ActPos >= Job[i].Target - para.TargetPosWindow
									AND NcToPlc.ActPos <= Job[i].Target + para.TargetPosWindow ;

		Job[i].InPosWindow	:= NcToPlc.ActPos >= Job[i].Target - para.PosRangeWindow
									AND NcToPlc.ActPos <= Job[i].Target + para.PosRangeWindow;
	END_IF
	
	IF Job[i].InTarget 
	THEN
		CheckTargetPos		:= i;
	END_IF
END_FOR
END_METHOD

PROPERTY PUBLIC optEnableCyclicCheckTargetPos : BOOL
GET
optEnableCyclicCheckTargetPos := Options.0;
END_GET
SET
Options.0 := optEnableCyclicCheckTargetPos;
END_SET
END_PROPERTY

METHOD PUBLIC startMotion : BOOL
VAR_INPUT
	Execute			:	BOOL;
	JobID			:	int ;
END_VAR
THIS^.JobID		:= Jobid;

IF JobID >= MIN_JOB AND JobId <= MAX_JOB
THEN
	CheckTargetPos();
//	startName				:= Job[Jobid].name;
	Motion.Fnc 				:= Job[Jobid].Fnc;
	Motion.BufferMode 		:= Job[Jobid].BufferMode;
	Motion.Direction 		:= Job[Jobid].Direction;
	Motion.Target 			:= Job[Jobid].Target;
	Motion.Velo 			:= Job[Jobid].Velo;
	Admin.Override 			:= Job[Jobid].Override;
	Motion.Acc		 		:= Job[Jobid].Acc;
	Motion.Dec				:= Job[Jobid].Dec;
	Motion.Jerk	 			:= Job[Jobid].Jerk;
	MOtion.Execute			:= Execute;
	StartMotion				:= TRUE;
ELSE
	StartMotion				:= FALSE;
END_IF
END_METHOD

END_FUNCTION_BLOCK

// POUs/Motion/TF5100-NCI/01_Main/NCI_REF
{attribute 'no_check'}
FUNCTION_BLOCK NCI_REF
VAR_INPUT
	PlcToNci										AT %Q*	: PLCTONC_NCICHANNEL_REF;	//link PLC to NC
END_VAR                             				
VAR_OUTPUT                          	
	NciToPlc										AT %I*	: NCTOPLC_NCICHANNEL_REF;	//link NC to PLC

(* Extrabits out of the struct *)
	ItpRunning												:	BOOL := FALSE;	//Interpreter is running
	ItpGroupActive											:	BOOL;			//Interpreter group is active -> Axes group build 			
	GrpCnfg													:	NCI_EXT3DGROUP;	//Group configuration
	                                    					
(* ChnState *******************)        					
	IsItpChn												:	BOOL := FALSE;	//TRUE when it is interpreter channel
	IsEStopRequested										:	BOOL := FALSE;	//TRUE when EStop is requested
	IsFeedFromBackupList									:	BOOL := FALSE;	//TRUE when parameter feed comes from backup list 
	IsMovingBackward										:	BOOL := FALSE;	//TRUE when moving forward
	
(* configurated parameters of the cyclic channel *)
	PathRestWay												:	LREAL;	//remaining arc length on the current path segment
	CurrentPathSetVelo										:	LREAL;	//current path set velocity
                                        					
	SAFStatus												:	UDINT;	//SAF state
	SAFEintraege											:	UDINT;	//current number of SAF entries/tasks
	SVBStatus												:	UDINT;	//SVB state
	SVBEintraege											:	UDINT;	//current number of SVB entries/tasks
	MemLastBlockNo											:	UDINT;	//contains last block number
END_VAR
VAR
	(* NciToPlc channel extend *)
	SetCyclicLrealOffsets									:	ItpSetCyclicLRealOffsets;
	SetCyclicLrealOffsetsDone								:	BOOL;
	SetCyclicUdintOffsets									:	ItpSetCyclicUdintOffsets;
	SetCyclicUdintOffsetsDone								:	BOOL;
	
END_VAR

;

METHOD readStatus : BOOL 
VAR_INPUT
END_VAR
(* NCI Status lesen															*)
(****************************************************************************)

(****************************************************************************)
(* 4 LReal variables to configurate the interface cyclely					*)
(****************************************************************************)
	IF SetCyclicLRealOffsets.bExecute AND NOT SetCyclicLRealOffsets.bBusy
	THEN
		SetCyclicLRealOffsetsDone := NOT SetCyclicLRealOffsets.bErr;
	END_IF

	IF NOT SetCyclicLRealOffsetsDone
	THEN
		SetCyclicLRealOffsets(
			bExecute			:= NciToPlc.ChnId <> 0 AND NOT SetCyclicLRealOffsetsDone AND NOT SetCyclicLRealOffsets.bErr,
			tTimeOut			:= DEFAULT_ADS_TIMEOUT,
			nIndexOffsetParam1	:= 16#500, (* Bahnrestweg (verbleibende Bogenlaenge) auf dem aktuellen Bahnsegment *)
			nIndexOffsetParam2	:= 16#502 , (* aktuelle Bahnsollgeschwindigkeit *)
			nIndexOffsetParam3	:= ,
			nIndexOffsetParam4	:= ,
			sNciToPlc			:= NciToPlc,
			bBusy				=> ,
			bErr				=> ,
			nErrId				=> );
	END_IF

	(* reading date *)
	PathRestWay												:= NciToPlc.DoubleParams[0];	
	CurrentPathSetVelo										:= NciToPlc.DoubleParams[1];	
	//														:= NciToPlc.DoubleParams[2];	
	//														:= NciToPlc.DoubleParams[0];	

(******************************************************************************)
(* 4 DINT variables cycliaclly das Zyklsiche Interface konfigurieren						*)
(******************************************************************************)
	IF SetCyclicUdintOffsets.bExecute 
	AND NOT SetCyclicUdintOffsets.bBusy
	THEN
		SetCyclicUdintOffsetsDone 							:= NOT SetCyclicUdintOffsets.bErr;
	END_IF

	IF NOT SetCyclicUdintOffsetsDone
	THEN
		SetCyclicUdintOffsets(
			bExecute			:= NciToPlc.ChnId <> 0 AND NOT SetCyclicUdintOffsetsDone AND NOT SetCyclicUdintOffsets.bErr,
			tTimeOut			:= DEFAULT_ADS_TIMEOUT,
			nIndexOffsetParam1	:= 16#4, (* Akt SVB Status 4  *)
			nIndexOffsetParam2	:= 16#5, (* Akt SAF Status -> Running 5 *)
			nIndexOffsetParam3	:= 16#B, (* Akt Anzahl SVB Eintraege B *)
			nIndexOffsetParam4	:= 16#C, (* Akt Anzahl SAF Eintraege C *)
			sNciToPlc			:= NciToPlc,
			bBusy				=> ,
			bErr				=> ,
			nErrId				=> );
	END_IF	

	(* Daten lesen *)
	SVBStatus												:= NciToPlc.IntParams[0];	
	SAFStatus												:= NciToPlc.IntParams[1];	
	SVBEintraege											:= NciToPlc.IntParams[2];	
	SAFEintraege											:= NciToPlc.IntParams[3];	
	
(******************************************************************************)
(* Interpreterstatus lesen																		*)
(******************************************************************************)
	ItpRunning 												:= NciToPlc.ItpState > NCI_INTERPRETER_READY
																	AND NciToPlc.ItpState <> NCI_INTERPRETER_ABORTED
																	OR SAFStatus > 2
																	OR SVBStatus > 2
																	OR SAFEintraege > 0
																	OR SVBEintraege > 0;
                                							
	IF NciToPlc.BlockNo > 0 
	AND MemLastBlockNo <> NciToPlc.BlockNo
	THEN
		MemLastBlockNo 	 									:= NciToPlc.BlockNo;
	END_IF                      							
	                            							
	GrpCnfg.nXAxisId										:= NciToPlc.AcsAxisIDs[0];
	GrpCnfg.nYAxisId										:= NciToPlc.AcsAxisIDs[1];
	GrpCnfg.nZAxisId										:= NciToPlc.AcsAxisIDs[2];
	GrpCnfg.nQ1AxisId										:= NciToPlc.AcsAxisIDs[3];
	GrpCnfg.nQ2AxisId										:= NciToPlc.AcsAxisIDs[4];
	GrpCnfg.nQ3AxisId										:=	NciToPlc.AcsAxisIDs[5];
	GrpCnfg.nQ4AxisId										:= NciToPlc.AcsAxisIDs[6];
	GrpCnfg.nQ5AxisId										:= NciToPlc.AcsAxisIDs[7];
                                							
	ItpGroupActive											:= GrpCnfg.nXAxisId <> 0
																	OR GrpCnfg.nYAxisId <> 0
																	OR GrpCnfg.nZAxisId <> 0
																	OR GrpCnfg.nQ1AxisId <> 0
																	OR GrpCnfg.nQ2AxisId <> 0
																	OR GrpCnfg.nQ3AxisId <> 0
																	OR GrpCnfg.nQ4AxisId <> 0
																	OR GrpCnfg.nQ5AxisId <> 0;
                                	
(******************************************************************************)
(* Channelstatus lesen																			*)
(******************************************************************************)
	IsItpChn												:= NciToPlc.ChnState.0;
	IsEStopRequested										:= NciToPlc.ChnState.8;
	IsFeedFromBackupList									:= NciToPlc.ChnState.10;
	IsMovingBackward										:= NciToPlc.ChnState.11;

	
(* ENUM ItpMode
	0x0	Defaultbelegung (Abwahl der übrigen Betriebsarten)
	0x1	Einzelsatzbetrieb im NC-Kern (Satzausführungstask/SAF)
	0x1000	reserviert
	0x2000	reserviert
	0x4000	Einzelsatzbetrieb im Interpreter
*)

(* ItpStatus
ITP_STATE_IDLE  The interpreter is in idle state when there is no NC program loaded as yet or when a group reset is being executed.
The interpreter also goes into idle state when a current program is stopped. In the case a group reset must be executed in order to prevent error 0x42C5. 
It is therefore recommended to execute a group reset after stopping via the PLC.
 
ITP_STATE_READY  After successful loading of an NC program, the interpreter is in ready state.
After a program has been successfully processed and exited, the interpreter goes into ready state. 
In the meantime, however, other states are accepted.  
 
ITP_STATE_ABORTED  Tritt während der Abarbeitung des NC Programms ein Laufzeitfehler auf, 
so geht der Interpreter in den Aborted eSTATE. Der eigentliche Fehlercode ist dem Kanal Status zu entnehmen.  

ITP_STATE_SINGLESTOP  If a run time error occurs during the processing of an NC program, the interpreter goes into aborted state. The actual error code is given in Channel Status.
 
NCI_INTERPRETER_INITFAILED:	UDINT	:=	0;
NCI_INTERPRETER_IDLE:			UDINT	:=	1;
NCI_INTERPRETER_READY:			UDINT	:=	2;
NCI_INTERPRETER_STARTED:		UDINT	:=	3;
NCI_INTERPRETER_SCANNING:		UDINT	:=	4;
NCI_INTERPRETER_RUNNING:		UDINT	:=	5;
NCI_INTERPRETER_STAY_RUNNING:	UDINT	:=	6;
NCI_INTERPRETER_WRITETABLE:		UDINT	:=	7;
NCI_INTERPRETER_SEARCHLINE:		UDINT	:=	8;
NCI_INTERPRETER_END:			UDINT	:=	9;
NCI_INTERPRETER_SINGLESTOP:		UDINT	:=	10;
NCI_INTERPRETER_ABORTING:		UDINT	:=	11;
NCI_INTERPRETER_ABORTED:		UDINT	:=	12;
NCI_INTERPRETER_FAULT:			UDINT	:=	13;
NCI_INTERPRETER_RESET:			UDINT	:=	14;
NCI_INTERPRETER_STOP:			UDINT := 15;
NCI_INTERPRETER_WAITFUNC:		UDINT	:=	16;
NCI_INTERPRETER_FLUSHBUFFERS:	UDINT	:=	17;

*)

	readStatus											:= TRUE;
(******************************************************************)
END_METHOD

END_FUNCTION_BLOCK

// POUs/Motion/TF5100-NCI/01_Main/NciAdmin
{attribute 'no_check'}
//NCI group administration - Build/Reconfig group via Enable input, activate EStop and StepOn after releasing EStop input
//based on Tc2_NCI library
FUNCTION_BLOCK NciAdmin
VAR_INPUT
	ResetAdmin												:	BOOL := FALSE; (* Reset Nci group *)
	Enable													:	BOOL := FALSE; (* TRUE = Build Group / FALSE = Reconfig Group *)
	EStop													:	BOOL := FALSE; (* TRUE = EStop / FALSE = StepOn *)
	SingleBlockMode											:	E_ItpSingleBlockMode := ItpSingleBlockOff; (* Operation mode for single set:
																											 	ItpSingleBlockOff: single set off
																											 	ItpSingleBlockNck: single set in the NC kernel 
																												ItpSingleBlockIntp: single set in the interpreter *)
	InSingleBlockTrigNext									:	BOOL	:= FALSE;
	GrpCnfg													:	NCI_EXT3DGROUP;
	Override												:	LREAL := 0.0; //0.0-100.0%
	SpindleOvr												:	LREAL := 0.0; //0.0-100.0%
	rNCIRef													:	REFERENCE TO NCI_REF := 0;
END_VAR
VAR_IN_OUT
END_VAR
VAR_OUTPUT
	InGroup													:	BOOL; 
	Busy													:	BOOL;
	Done													:	BOOL;
	Error													:	BOOL;
{attribute 'displaymode':='hex'}
	ErrorID													:	UDINT;
	ErrorText												:	STRING(40);
END_VAR
VAR
(* Zwischenspeicher **************************************************************************)
	MemDone													:	BOOL;
	MemFnc													:	INT := 0;

(* Instanzierung der MC Bausteine *******************************************************)
	ItpSingleBlock											:	ItpSingleBlock := (tTimeOut	:= DEFAULT_ADS_TIMEOUT);
	CfgBuildExt3DGroup										:	CfgBuildExt3DGroup := (tTimeOut	:= DEFAULT_ADS_TIMEOUT);
	CfgReconfigGroup										:	CfgReconfigGroup := (tTimeOut	:= DEFAULT_ADS_TIMEOUT);
	ItpResetEx2												:	ItpResetEx2 := (tTimeOut	:= DEFAULT_ADS_TIMEOUT);
	ItpEStopEx												:	ItpEStopEx := (tTimeOut	:= DEFAULT_ADS_TIMEOUT);
	ItpStepOnAfterEStopEx									:	ItpStepOnAfterEStopEx := (tTimeOut	:= DEFAULT_ADS_TIMEOUT);

(* Dummy  **********************************************************)
	Dummy 	: BOOL;
END_VAR

	(* NCI group administration															*)
	(************************************************************************************)

(* verify reference ***********************************************************************)
IF NOT __ISVALIDREF(rNCIRef) 
THEN
	Busy													:= NOT Error;
	ErrorId													:= E_AdsErr.DEVICE_INVALIDPARM;
	Error													:= TRUE;
	Done													:= FALSE;
	InGroup													:= FALSE;
	ErrorText												:= 'Reference to rNCIRef invalid (0)';
	RETURN;
END_IF

(* reading axis-status from NCtoPLC-channel *************************************************)
	rNCIRef.ReadStatus();

(* writing override into the NC-interface ***************************************************)
	rNCIRef.PlcToNci.ChnAxesOvr 							:= LREAL_TO_DWORD(LIMIT(0.0,Override,100.0) * 10000.0 );
	rNCIRef.PlcToNci.ChnSpindleOvr							:= LREAL_TO_DWORD(LIMIT(0.0,SpindleOvr,100.0) * 10000.0 );

